VAR_TEMP
  EStopOK : BOOL ;	//auxiliary flag
  CIP : BOOL ;	//CIP Program Selected
  xTmp : BOOL ;	//Temporary Bool(free for general use)
  UnitNo : INT ;	//unit number
  UnitFB : INT ;	//unit expansion FB number
  rTmp : REAL ;	//Temporary REAL (free for general use)
  iTmp : INT ;	//Temporary INT (free for general use)
  dTmp : DINT ;	//Temporary DINT (free for general use)
END_VAR
BEGIN
NETWORK
TITLE =general

      CLR   ;
      =     #xTmp;
      =     #EStopOK;

      L     DB1950.DBW    0;
      T     #UnitNo;
      L     DB1950.DBW    2;
      T     #UnitFB;

NETWORK
TITLE =Universal value

      NOP   0;
// unv001 UnV 001 Process Status
      CALL FC    27 (
           UnitNo                   := #UnitNo,
           UnVRec                   := DB2955.unv001,
           ValExt                   := DB2955.DBD  234);

// unv002 UnV 002 Universal Value 02
      CALL FC    27 (
           UnitNo                   := #UnitNo,
           UnVRec                   := DB2955.unv002,
           ValExt                   := DB2955.DBD  362);

// RK2_KreisNr UnV 003 Circuit Number
      CALL FC    27 (
           UnitNo                   := #UnitNo,
           UnVRec                   := DB2955.RK2_KreisNr,
           ValExt                   := DB2955.DBD  490);

// RK2_Medium UnV 004 0=NIX 1=Wasser 2=Heißwasser 3=Lauge 4=Säure 5=Desi
      CALL FC    27 (
           UnitNo                   := #UnitNo,
           UnVRec                   := DB2955.RK2_Medium,
           ValExt                   := DB2955.DBD  618);

NETWORK
TITLE =special inputs

      NOP   0;
// GOA_RR2 SpI 001 GOA_RR2 Schwenkbogen Befüllblock nach RR2
      CALL FC    14 (
           UnitNo                   := #UnitNo,
           SpIRec                   := DB2951.GOA_RR2,
           SpIBit                   := I    312.0);

// RM_NI_RR2K1 SpI 002 Handklappe im Rücklauf CIP 2 hinter Befüllblock
      CALL FC    14 (
           UnitNo                   := #UnitNo,
           SpIRec                   := DB2951.RM_NI_RR2K1,
           SpIBit                   := I    312.2);

// GOA_RV2K1 SpI 003 RV2K1
      CALL FC    14 (
           UnitNo                   := #UnitNo,
           SpIRec                   := DB2951.GOA_RV2K1,
           SpIBit                   := I    276.0);

// GOA_RV2K2 SpI 004 RV2K2 zur KEG Anlage
      CALL FC    14 (
           UnitNo                   := #UnitNo,
           SpIRec                   := DB2951.GOA_RV2K2,
           SpIBit                   := I    276.1);

NETWORK
TITLE =messages

      NOP   0;
// msg001 Msg 001 Message 01
      CALL FC    16 (
           UnitNo                   := #UnitNo,
           MsgRec                   := DB2957.msg001,
           MsgBit                   := DB2957.DBX   82.7);

// msg002 Msg 002 Message 02
      CALL FC    16 (
           UnitNo                   := #UnitNo,
           MsgRec                   := DB2957.msg002,
           MsgBit                   := DB2957.DBX  142.7);

NETWORK
TITLE =unit supply

      UC    FB [#UnitFB];

NETWORK
TITLE =FW_RK1
// Act 003
// Box           : Ventilinsel 4
// Input address : I335.7
// Output address: Q335.7
      CALL FC    70 (
           UnitNo                   := #UnitNo,
           ActRec                   := DB2950.FW_RK1,
           Typ                      := 23,
           FBa                      := I    335.7,
           FBa2                     := #xTmp,
           Out                      := Q    335.7);

NETWORK
TITLE =RV2_RW
// Act 004
// Box           : VSRVK1..3
// Input address : I82.1
// Output address: Q82.1
      CALL FC    70 (
           UnitNo                   := #UnitNo,
           ActRec                   := DB2950.RV2_RW,
           Typ                      := 1,
           FBa                      := #xTmp,
           FBa2                     := I     82.1,
           Out                      := Q     82.1);

NETWORK
TITLE =RV2V1  KEG/A14 KZE
// Act 006
// Box           : VS2-BB
// Output address: Q311.1
      CALL FC    70 (
           UnitNo                   := #UnitNo,
           ActRec                   := DB2950.RV2V1,
           Typ                      := 0,
           FBa                      := #xTmp,
           FBa2                     := #xTmp,
           Out                      := Q    311.1);

NETWORK
TITLE =RV2_RS  Ventil zum Gully beim spülen vom Tank
// Act 007
// Box           : Ventilinsel 4
// Input address : I337.3
// Output address: Q337.3
      CALL FC    70 (
           UnitNo                   := #UnitNo,
           ActRec                   := DB2950.RV2_RS,
           Typ                      := 1,
           FBa                      := #xTmp,
           FBa2                     := I    337.3,
           Out                      := Q    337.3);

END_FUNCTION_BLOCK

FUNCTION_BLOCK FB 1951
TITLE =U095: CIP 2 Distribution
FAMILY : BOTEC_F1
NAME : UniE
VERSION : 1.2


VAR_TEMP
  CIP : BOOL ;	//CIP active
  UNIM : BOOL ;	//Unit Not In Maintenance
  GenRel : BOOL ;	//general OK (emergency and maintenance OK)
  EStopOK : BOOL ;	//emergency OK
  UnitNo : INT ;	//unit number
  xTmp : BOOL ;	//Temporary Bool
  iTmp : INT ;	//Temporary INT
  rTmp : REAL ;	//Temporary REAL
  dTmp : DINT ;	//Temporary DINT (free for general use)
  RetValInt : INT ;	//return value
END_VAR
BEGIN
NETWORK
TITLE =General

      SET   ;
// Simulation ---------------------------------------------------------------
      A     DB1951.DBX 1357.7;
      CC    FB  1959; // "U095Sim"
      A     DB1951.DBX   17.3;
      =     DB1951.DBX 1357.7; //Help bit for simulation

// get unit number ----------------------------------------------------------
      L     DB1950.DBW    0;
      T     #UnitNo;

// CIP ----------------------------------------------------------------------
      L     DB1951.DBD   54;
      L     0;
      <D    ;
      =     #CIP;

// emergency OK -------------------------------------------------------------
      A     DB1955.DBX   27.0; //Emergency Stop OK
      =     #EStopOK;

// Write Unit in Maintenance ------------------------------------------------

      AN    DB1951.DBX   69.7;
      =     #UNIM;

// emergency and maintenance OK ---------------------------------------------
      A     #EStopOK;
      A     #UNIM;
      =     #GenRel;

// communication ------------------------------------------------------------
      UC    FB  1955; // U095Com

NETWORK
TITLE =Universal Value

      NOP   0;

// ----------------------------------------------------------
// unv001 Process Status
// ----------------------------------------------------------
// process value to UnV
//      L     0.000000e+000
//      T     "U095UnVD".unv001.ValExt

// ----------------------------------------------------------
// unv002 Universal Value 02
// ----------------------------------------------------------
// process value to UnV
//      L     0.000000e+000
//      T     "U095UnVD".unv002.ValExt

// ----------------------------------------------------------
// RK2_KreisNr Circuit Number
// ----------------------------------------------------------
// process value to UnV
//      L     0.000000e+000
//      T     "U095UnVD".RK2_KreisNr.ValExt

// ----------------------------------------------------------
// RK2_Medium 0=NIX 1=Wasser 2=Heißwasser 3=Lauge 4=Säure 5=Desi
// ----------------------------------------------------------
// process value to UnV
//      L     0.000000e+000
//      T     "U095UnVD".RK2_Medium.ValExt

NETWORK
TITLE =Special Input

      NOP   0;

// ----------------------------------------------------------
// GOA_RR2 GOA_RR2 Schwenkbogen Befüllblock nach RR2
// ----------------------------------------------------------
//      SET
//      =     "U095SpID".GOA_RR2.EAl
//      =     "U095SpID".GOA_RR2.Pre

// ----------------------------------------------------------
// RM_NI_RR2K1 Handklappe im Rücklauf CIP 2 hinter Befüllblock
// ----------------------------------------------------------
      SET   ;
      =     DB2951.DBX  141.4;
      =     DB2951.DBX  141.5;

// ----------------------------------------------------------
// GOA_RV2K1 RV2K1
// ----------------------------------------------------------
      SET   ;
      =     DB2951.DBX  201.4;
      =     DB2951.DBX  201.5;

// ----------------------------------------------------------
// GOA_RV2K2 RV2K2 zur KEG Anlage
// ----------------------------------------------------------
      SET   ;
      =     DB2951.DBX  261.4;
      =     DB2951.DBX  261.5;

NETWORK
TITLE =Messages

      NOP   0;

// ----------------------------------------------------------
// msg001 Message 01
// ----------------------------------------------------------
      SET   ;
      R     DB2957.DBX   80.7;
      =     DB2957.DBX   81.4;

      CLR   ;
      =     DB2957.DBX   82.7;

// ----------------------------------------------------------
// msg002 Message 02
// ----------------------------------------------------------
      SET   ;
      R     DB2957.DBX  140.7;
      =     DB2957.DBX  141.4;

      CLR   ;
      =     DB2957.DBX  142.7;

NETWORK
TITLE =Sequence organisation

      CLR   ;
      =     M    122.2;

// SFM supply ----------------------------------------------------------------

// CIP Counter
//      CALL  "V2S"
//       UnitNo      :=#UnitNo
//       Value       :="U095ComD".Own.Real07
//       Enable      :=TRUE
//       Down        :=FALSE
//       OriginDetect:=0.000000e+000
//       MaxDiffPS   :=1.000000e+000
//       SFMRec      :="U095SeqD".Seq.SFM[15]
//       ValueOld    :="U095SeqD".Seq.User.Real15

// sequencer ----------------------------------------------------------------
      A     DB1953.DBX   43.1;
      S     DB1953.DBX   97.3;

      CALL FC    40 (
           UnitNo                   := #UnitNo);

NETWORK
TITLE =Auto / Manual

      SET   ;
      AN    M    122.2;
      JC    MODE;
      AN    M    120.1;
      =     DB2950.DBX  265.4;
      =     DB2950.DBX  345.4;
      =     DB2950.DBX  505.4;
      =     DB2950.DBX  585.4;


MODE: SET   ;


NETWORK
TITLE =FW_RK1
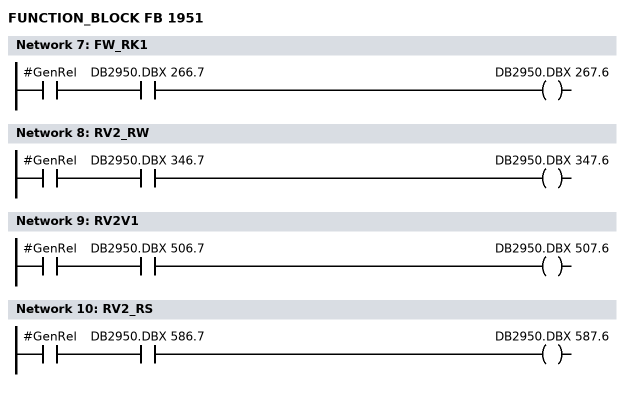

      A     #GenRel;
      A     DB2950.DBX  266.7;
      =     DB2950.DBX  267.6;
NETWORK
TITLE =RV2_RW

      A     #GenRel;
      A     DB2950.DBX  346.7;
      =     DB2950.DBX  347.6;

NETWORK
TITLE =RV2V1

      A     #GenRel;
      A     DB2950.DBX  506.7;
      =     DB2950.DBX  507.6;
NETWORK
TITLE =RV2_RS


      A     #GenRel;
      A     DB2950.DBX  586.7;
      =     DB2950.DBX  587.6;
END_FUNCTION_BLOCK

FUNCTION_BLOCK FB 1960
TITLE =U096: CIP 3 Distribution
FAMILY : BOTEC_F1
NAME : UniA
VERSION : 2.1


VAR_TEMP
  EStopOK : BOOL ;	//auxiliary flag
  CIP : BOOL ;	//CIP Program Selected
  xTmp : BOOL ;	//Temporary Bool(free for general use)
  UnitNo : INT ;	//unit number
  UnitFB : INT ;	//unit expansion FB number
  rTmp : REAL ;	//Temporary REAL (free for general use)
  iTmp : INT ;	//Temporary INT (free for general use)
  dTmp : DINT ;	//Temporary DINT (free for general use)
END_VAR
BEGIN
NETWORK
TITLE =general

      CLR   ;
      =     #xTmp;
      =     #EStopOK;

      L     DB1960.DBW    0;
      T     #UnitNo;
      L     DB1960.DBW    2;
      T     #UnitFB;

NETWORK
TITLE =Universal value

      NOP   0;
// unv001 UnV 001 Process Status
      CALL FC    27 (
           UnitNo                   := #UnitNo,
           UnVRec                   := DB2965.unv001,
           ValExt                   := DB2965.DBD  234);

// unv002 UnV 002 Universal Value 02
      CALL FC    27 (
           UnitNo                   := #UnitNo,
           UnVRec                   := DB2965.unv002,
           ValExt                   := DB2965.DBD  362);

// RK3_KreisNr UnV 003 Circuit Number
      CALL FC    27 (
           UnitNo                   := #UnitNo,
           UnVRec                   := DB2965.RK3_KreisNr,
           ValExt                   := DB2965.DBD  490);

// RK3_Medium UnV 004 0=NIX 1=Wasser 2=Heißwasser 3=Lauge 4=Säure 5=Desi
      CALL FC    27 (
           UnitNo                   := #UnitNo,
           UnVRec                   := DB2965.RK3_Medium,
           ValExt                   := DB2965.DBD  618);

NETWORK
TITLE =special inputs

      NOP   0;
// RK3_I_Bereit SpI 001 Das Reinigungs Programm ist gestartet und läuft "1"= Läuft  "0"=AUS
      CALL FC    14 (
           UnitNo                   := #UnitNo,
           SpIRec                   := DB2961.RK3_I_Bereit,
           SpIBit                   := DB304.DBX   30.0);

// RK3_I_VL_Ein SpI 002 Medium wird angefordert (Reinigungs Vorlauf EIN) "1"=VorlaufPumpe an "0"AUS
      CALL FC    14 (
           UnitNo                   := #UnitNo,
           SpIRec                   := DB2961.RK3_I_VL_Ein,
           SpIBit                   := DB304.DBX   30.1);

// RK3_I_RL_Ein SpI 003 Medium wird zurückgepumpt "1" RücklaufPumpe an "0"=AUS
      CALL FC    14 (
           UnitNo                   := #UnitNo,
           SpIRec                   := DB2961.RK3_I_RL_Ein,
           SpIBit                   := DB304.DBX   30.2);

// RK3_I_Leer SpI 004 Der zu Reinigende Anlagenteil ist leer."1"=leer "0"=nicht leer
      CALL FC    14 (
           UnitNo                   := #UnitNo,
           SpIRec                   := DB2961.RK3_I_Leer,
           SpIBit                   := DB304.DBX   30.3);

// RK3_I_Stop SpI 005 Stop interner Fehler Pumpen anhalten Reinigungszeit anhalten "1" STOP  "0"= OK
      CALL FC    14 (
           UnitNo                   := #UnitNo,
           SpIRec                   := DB2961.RK3_I_Stop,
           SpIBit                   := DB304.DBX   30.4);

// RK3_I_SK_RM SpI 006 Bypassventil ist angesteuert und offen
      CALL FC    14 (
           UnitNo                   := #UnitNo,
           SpIRec                   := DB2961.RK3_I_SK_RM,
           SpIBit                   := DB304.DBX   30.7);

NETWORK
TITLE =messages

      NOP   0;
// msg001 Msg 001 Message 01
      CALL FC    16 (
           UnitNo                   := #UnitNo,
           MsgRec                   := DB2967.msg001,
           MsgBit                   := DB2967.DBX   82.7);

// msg002 Msg 002 Message 02
      CALL FC    16 (
           UnitNo                   := #UnitNo,
           MsgRec                   := DB2967.msg002,
           MsgBit                   := DB2967.DBX  142.7);

NETWORK
TITLE =unit supply

      UC    FB [#UnitFB];

NETWORK
TITLE =RV3_ST
// Act 004
// Box           : VSRVK1..3
// Input address : I82.2
// Output address: Q82.2
      CALL FC    70 (
           UnitNo                   := #UnitNo,
           ActRec                   := DB2960.RV3_ST,
           Typ                      := 1,
           FBa                      := #xTmp,
           FBa2                     := I     82.2,
           Out                      := Q     82.2);

NETWORK
TITLE =K3_VNI_RSTP  STOP TU AN VNI MELDEN
// Act 004
// Box           : S8 U8.2
// Output address: Q42.0
      CALL FC    70 (
           UnitNo                   := #UnitNo,
           ActRec                   := DB2960.K3_VNI_RSTP,
           Typ                      := 0,
           FBa                      := #xTmp,
           FBa2                     := #xTmp,
           Out                      := Q     42.0);

NETWORK
TITLE =K3_VNI_RMW  MEDIENWECHSEL AN VNI MELDEN
// Act 005
// Box           : S8 U8.2
// Output address: Q42.1
      CALL FC    70 (
           UnitNo                   := #UnitNo,
           ActRec                   := DB2960.K3_VNI_RMW,
           Typ                      := 0,
           FBa                      := #xTmp,
           FBa2                     := #xTmp,
           Out                      := Q     42.1);

NETWORK
TITLE =K3_VNI_REND  ENDE MELDUNG AN VNI
// Act 006
// Box           : S8 U8.2
// Output address: Q42.2
      CALL FC    70 (
           UnitNo                   := #UnitNo,
           ActRec                   := DB2960.K3_VNI_REND,
           Typ                      := 0,
           FBa                      := #xTmp,
           FBa2                     := #xTmp,
           Out                      := Q     42.2);

NETWORK
TITLE =K3_VNI_RHL  MELDUNG HEISSLAUGE AN VNI
// Act 007
// Box           : S8 U8.2
// Output address: Q42.3
      CALL FC    70 (
           UnitNo                   := #UnitNo,
           ActRec                   := DB2960.K3_VNI_RHL,
           Typ                      := 0,
           FBa                      := #xTmp,
           FBa2                     := #xTmp,
           Out                      := Q     42.3);

NETWORK
TITLE =K3_VNI_RBTR  BETRIEBSMELDUNG CIP AN VNI
// Act 008
// Box           : S8 U8.2
// Output address: Q42.4
      CALL FC    70 (
           UnitNo                   := #UnitNo,
           ActRec                   := DB2960.K3_VNI_RBTR,
           Typ                      := 0,
           FBa                      := #xTmp,
           FBa2                     := #xTmp,
           Out                      := Q     42.4);

NETWORK
TITLE =K3_VNI_WASSER_OK  WASSER OK AN VNI
// Act 009
// Box           : S8 U8.2
// Output address: Q42.5
      CALL FC    70 (
           UnitNo                   := #UnitNo,
           ActRec                   := DB2960.K3_VNI_WASSER_OK,
           Typ                      := 0,
           FBa                      := #xTmp,
           FBa2                     := #xTmp,
           Out                      := Q     42.5);

NETWORK
TITLE =RK3_Bereit  Die CIP Station hat gestatet "0"=AUS "1"=gestartet
// Act 010
// Box           : Sirup
// Output address: DB_SEND_DOEHLER.RK3.Bereit
      CALL FC    70 (
           UnitNo                   := #UnitNo,
           ActRec                   := DB2960.RK3_Bereit,
           Typ                      := 0,
           FBa                      := #xTmp,
           FBa2                     := #xTmp,
           Out                      := DB404.DBX   30.0);

NETWORK
TITLE =RK3_Stop  Stop Pumpen anhalten "0"Ok" 1"=Stop
// Act 011
// Box           : Sirup
// Output address: DB_SEND_DOEHLER.RK3.Stop
      CALL FC    70 (
           UnitNo                   := #UnitNo,
           ActRec                   := DB2960.RK3_Stop,
           Typ                      := 0,
           FBa                      := #xTmp,
           FBa2                     := #xTmp,
           Out                      := DB404.DBX   30.1);

NETWORK
TITLE =RK3_MED  Medienwechsel der CIP
// Act 012
// Box           : Sirup
// Output address: DB_SEND_DOEHLER.RK3.MED
      CALL FC    70 (
           UnitNo                   := #UnitNo,
           ActRec                   := DB2960.RK3_MED,
           Typ                      := 0,
           FBa                      := #xTmp,
           FBa2                     := #xTmp,
           Out                      := DB404.DBX   30.2);

NETWORK
TITLE =RK3_ENDE  Ende der Reinigung
// Act 013
// Box           : Sirup
// Output address: DB_SEND_DOEHLER.RK3.ENDE
      CALL FC    70 (
           UnitNo                   := #UnitNo,
           ActRec                   := DB2960.RK3_ENDE,
           Typ                      := 0,
           FBa                      := #xTmp,
           FBa2                     := #xTmp,
           Out                      := DB404.DBX   30.3);

NETWORK
TITLE =RK3_Bypass  CIP Bypass
// Act 014
// Box           : Sirup
// Output address: DB_SEND_DOEHLER.RK3.Bypass
      CALL FC    70 (
           UnitNo                   := #UnitNo,
           ActRec                   := DB2960.RK3_Bypass,
           Typ                      := 0,
           FBa                      := #xTmp,
           FBa2                     := #xTmp,
           Out                      := DB404.DBX   30.4);

NETWORK
TITLE =SR1_RR3  SR1 RR3 CIP Rücklaufventil RR3SR1
// Act 015
// Box           : VS-RRA
// Input address : I200.7
// Output address: Q200.7
      CALL FC    70 (
           UnitNo                   := #UnitNo,
           ActRec                   := DB2960.SR1_RR3,
           Typ                      := 1,
           FBa                      := #xTmp,
           FBa2                     := I    200.7,
           Out                      := Q    200.7);

NETWORK
TITLE =SR2_RR3  SR2 RR3 CIP Rücklaufventil RR3SR2
// Act 016
// Box           : VS-RRA
// Input address : I201.1
// Output address: Q201.1
      CALL FC    70 (
           UnitNo                   := #UnitNo,
           ActRec                   := DB2960.SR2_RR3,
           Typ                      := 1,
           FBa                      := #xTmp,
           FBa2                     := I    201.1,
           Out                      := Q    201.1);

NETWORK
TITLE =RV3_RS  Ventil zum Gully beim spülen vom Tank
// Act 019
// Box           : Ventilinsel 4
// Input address : I337.4
// Output address: Q337.4
      CALL FC    70 (
           UnitNo                   := #UnitNo,
           ActRec                   := DB2960.RV3_RS,
           Typ                      := 1,
           FBa                      := #xTmp,
           FBa2                     := I    337.4,
           Out                      := Q    337.4);

END_FUNCTION_BLOCK

FUNCTION_BLOCK FB 1961
TITLE =U096: CIP 3 Distribution
FAMILY : BOTEC_F1
NAME : UniE
VERSION : 1.2


VAR_TEMP
  CIP : BOOL ;	//CIP active
  UNIM : BOOL ;	//Unit Not In Maintenance
  GenRel : BOOL ;	//general OK (emergency and maintenance OK)
  EStopOK : BOOL ;	//emergency OK
  UnitNo : INT ;	//unit number
  xTmp : BOOL ;	//Temporary Bool
  iTmp : INT ;	//Temporary INT
  rTmp : REAL ;	//Temporary REAL
  dTmp : DINT ;	//Temporary DINT (free for general use)
  RetValInt : INT ;	//return value
END_VAR
BEGIN
NETWORK
TITLE =General

      SET   ;
// Simulation ---------------------------------------------------------------
      A     DB1961.DBX 1357.7;
      CC    FB  1969; // "U096Sim"
      A     DB1961.DBX   17.3;
      =     DB1961.DBX 1357.7; //Help bit for simulation

// get unit number ----------------------------------------------------------
      L     DB1960.DBW    0;
      T     #UnitNo;

// CIP ----------------------------------------------------------------------
      L     DB1961.DBD   54;
      L     0;
      <D    ;
      =     #CIP;

// emergency OK -------------------------------------------------------------
      A     DB1965.DBX   27.0; //Emergency Stop OK
      =     #EStopOK;

// Write Unit in Maintenance ------------------------------------------------

      AN    DB1961.DBX   69.7;
      =     #UNIM;

// emergency and maintenance OK ---------------------------------------------
      A     #EStopOK;
      A     #UNIM;
      =     #GenRel;

// communication ------------------------------------------------------------
      UC    FB  1965; // U096Com

NETWORK
TITLE =Universal Value

      NOP   0;

// ----------------------------------------------------------
// unv001 Process Status
// ----------------------------------------------------------
// process value to UnV
//      L     0.000000e+000
//      T     "U096UnVD".unv001.ValExt

// ----------------------------------------------------------
// unv002 Universal Value 02
// ----------------------------------------------------------
// process value to UnV
//      L     0.000000e+000
//      T     "U096UnVD".unv002.ValExt

// ----------------------------------------------------------
// RK3_KreisNr Circuit Number
// ----------------------------------------------------------
// process value to UnV
//      L     0.000000e+000
//      T     "U096UnVD".RK3_KreisNr.ValExt

// ----------------------------------------------------------
// RK3_Medium 0=NIX 1=Wasser 2=Heißwasser 3=Lauge 4=Säure 5=Desi
// ----------------------------------------------------------
// process value to UnV
//      L     0.000000e+000
//      T     "U096UnVD".RK3_Medium.ValExt

NETWORK
TITLE =Special Input

      NOP   0;

// ----------------------------------------------------------
// RK3_I_Bereit Das Reinigungs Programm ist gestartet und läuft "1"= Läuft  "0"=AUS
// ----------------------------------------------------------
      CLR   ;
      =     DB2961.DBX   81.4;
      =     DB2961.DBX   81.5;

// ----------------------------------------------------------
// RK3_I_VL_Ein Medium wird angefordert (Reinigungs Vorlauf EIN) "1"=VorlaufPumpe an "0"AUS
// ----------------------------------------------------------
      CLR   ;
      =     DB2961.DBX  141.4;
      =     DB2961.DBX  141.5;

// ----------------------------------------------------------
// RK3_I_RL_Ein Medium wird zurückgepumpt "1" RücklaufPumpe an "0"=AUS
// ----------------------------------------------------------
      CLR   ;
      =     DB2961.DBX  201.4;
      =     DB2961.DBX  201.5;

// ----------------------------------------------------------
// RK3_I_Leer Der zu Reinigende Anlagenteil ist leer."1"=leer "0"=nicht leer
// ----------------------------------------------------------
      CLR   ;
      =     DB2961.DBX  261.4;
      =     DB2961.DBX  261.5;

// ----------------------------------------------------------
// RK3_I_Stop Stop interner Fehler Pumpen anhalten Reinigungszeit anhalten "1" STOP  "0"= OK
// ----------------------------------------------------------
      CLR   ;
      =     DB2961.DBX  321.4;
      =     DB2961.DBX  321.5;

// ----------------------------------------------------------
// RK3_I_SK_RM Bypassventil ist angesteuert und offen
// ----------------------------------------------------------
      CLR   ;
      =     DB2961.DBX  381.4;
      =     DB2961.DBX  381.5;

NETWORK
TITLE =Messages

      NOP   0;

// ----------------------------------------------------------
// msg001 Message 01
// ----------------------------------------------------------
      SET   ;
      R     DB2967.DBX   80.7;
      =     DB2967.DBX   81.4;

      CLR   ;
      =     DB2967.DBX   82.7;

// ----------------------------------------------------------
// msg002 Message 02
// ----------------------------------------------------------
      SET   ;
      R     DB2967.DBX  140.7;
      =     DB2967.DBX  141.4;

      CLR   ;
      =     DB2967.DBX  142.7;

NETWORK
TITLE =Sequence organisation

      CLR   ;
      =     M    122.2;

// SFM supply ----------------------------------------------------------------

      CALL FC    29 (
           UnitNo                   := #UnitNo,
           Value                    := DB1965.DBD   54,
           Enable                   := TRUE,
           Down                     := FALSE,
           OriginDetect             := 0.000000e+000,
           MaxDiffPS                := 1.000000e+000,
           SFMRec                   := DB1961.Seq.SFM[15],
           ValueOld                 := DB1961.DBD 1418);

// sequencer ----------------------------------------------------------------
      A     DB1963.DBX   43.1;
      S     DB1963.DBX   97.3;

      CALL FC    40 (
           UnitNo                   := #UnitNo);

NETWORK
TITLE =Auto / Manual

      SET   ;
      AN    M    122.2;
      JC    MODE;
      AN    M    120.1;

// assign actuator mode
      AN    M    120.1;
      =     DB2960.DBX  185.4;
      =     DB2960.DBX  265.4;
      =     DB2960.DBX  345.4;
      =     DB2960.DBX  425.4;
      =     DB2960.DBX  505.4;
      =     DB2960.DBX  585.4;
      =     DB2960.DBX  665.4;
      =     DB2960.DBX  745.4;
      =     DB2960.DBX  825.4;
      =     DB2960.DBX  905.4;
      =     DB2960.DBX  985.4;
      =     DB2960.DBX 1065.4;
      =     DB2960.DBX 1145.4;
      =     DB2960.DBX 1225.4;
      =     DB2960.DBX 1305.4;
      =     DB2960.DBX 1545.4;

MODE: SET   ;

NETWORK
TITLE =RV3_ST
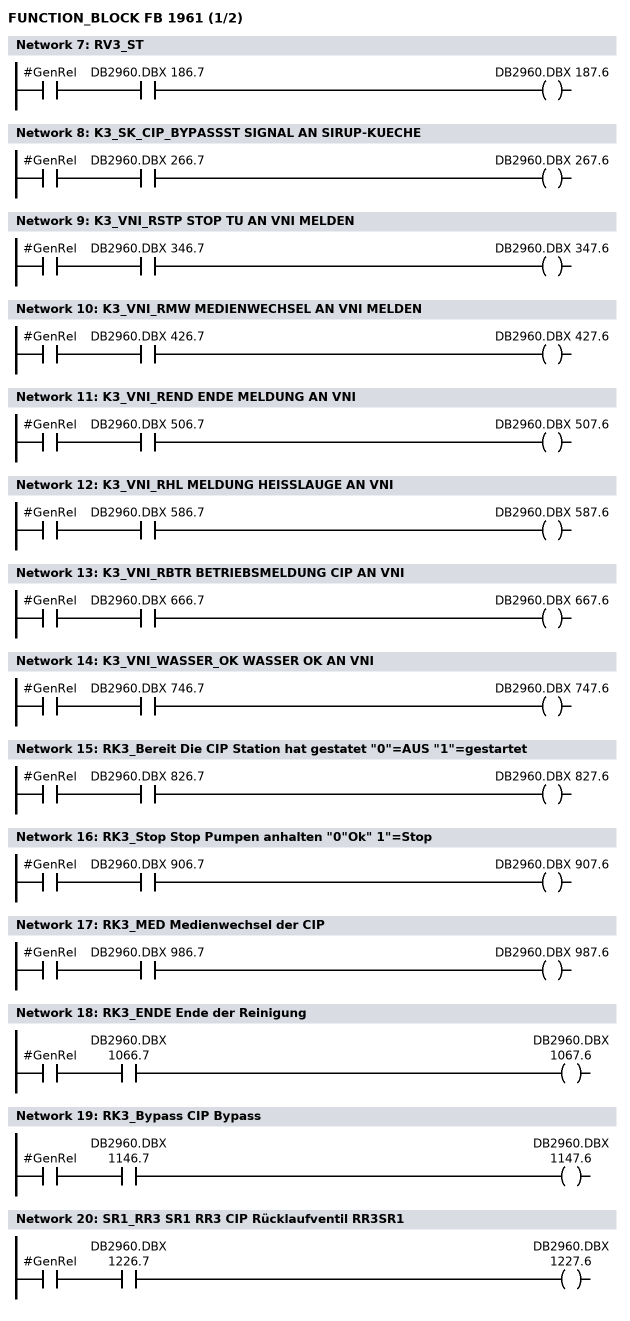

      A     #GenRel;
      A     DB2960.DBX  186.7;
      =     DB2960.DBX  187.6;
NETWORK
TITLE =K3_SK_CIP_BYPASSST SIGNAL AN SIRUP-KUECHE

      A     #GenRel;
      A     DB2960.DBX  266.7;
      =     DB2960.DBX  267.6;
NETWORK
TITLE =K3_VNI_RSTP STOP TU AN VNI MELDEN

      A     #GenRel;
      A     DB2960.DBX  346.7;
      =     DB2960.DBX  347.6;
NETWORK
TITLE =K3_VNI_RMW MEDIENWECHSEL AN VNI MELDEN

      A     #GenRel;
      A     DB2960.DBX  426.7;
      =     DB2960.DBX  427.6;
NETWORK
TITLE =K3_VNI_REND ENDE MELDUNG AN VNI

      A     #GenRel;
      A     DB2960.DBX  506.7;
      =     DB2960.DBX  507.6;
NETWORK
TITLE =K3_VNI_RHL MELDUNG HEISSLAUGE AN VNI

      A     #GenRel;
      A     DB2960.DBX  586.7;
      =     DB2960.DBX  587.6;
NETWORK
TITLE =K3_VNI_RBTR BETRIEBSMELDUNG CIP AN VNI

      A     #GenRel;
      A     DB2960.DBX  666.7;
      =     DB2960.DBX  667.6;
NETWORK
TITLE =K3_VNI_WASSER_OK WASSER OK AN VNI

      A     #GenRel;
      A     DB2960.DBX  746.7;
      =     DB2960.DBX  747.6;
NETWORK
TITLE =RK3_Bereit Die CIP Station hat gestatet "0"=AUS "1"=gestartet

      A     #GenRel;
      A     DB2960.DBX  826.7;
      =     DB2960.DBX  827.6;
NETWORK
TITLE =RK3_Stop Stop Pumpen anhalten "0"Ok" 1"=Stop

      A     #GenRel;
      A     DB2960.DBX  906.7;
      =     DB2960.DBX  907.6;
NETWORK
TITLE =RK3_MED Medienwechsel der CIP

      A     #GenRel;
      A     DB2960.DBX  986.7;
      =     DB2960.DBX  987.6;
NETWORK
TITLE =RK3_ENDE Ende der Reinigung

      A     #GenRel;
      A     DB2960.DBX 1066.7;
      =     DB2960.DBX 1067.6;
NETWORK
TITLE =RK3_Bypass CIP Bypass

      A     #GenRel;
      A     DB2960.DBX 1146.7;
      =     DB2960.DBX 1147.6;
NETWORK
TITLE =SR1_RR3 SR1 RR3 CIP Rücklaufventil RR3SR1

      A     #GenRel;
      A     DB2960.DBX 1226.7;
      =     DB2960.DBX 1227.6;
NETWORK
TITLE =SR2_RR3 SR2 RR3 CIP Rücklaufventil RR3SR2
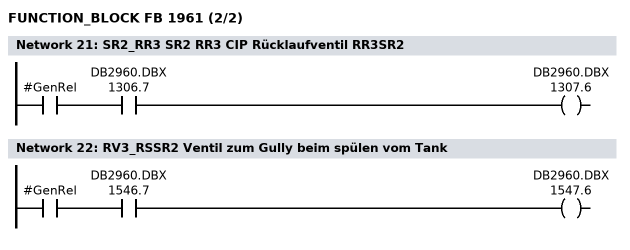

      A     #GenRel;
      A     DB2960.DBX 1306.7;
      =     DB2960.DBX 1307.6;
NETWORK
TITLE =RV3_RSSR2 Ventil zum Gully beim spülen vom Tank

      A     #GenRel;
      A     DB2960.DBX 1546.7;
      =     DB2960.DBX 1547.6;
END_FUNCTION_BLOCK

FUNCTION_BLOCK FB 1980
TITLE =U098: General Syrup Room
FAMILY : BOTEC_F1
NAME : UniA
VERSION : 2.1


VAR_TEMP
  EStopOK : BOOL ;	//auxiliary flag
  CIP : BOOL ;	//CIP Program Selected
  xTmp : BOOL ;	//Temporary Bool(free for general use)
  UnitNo : INT ;	//unit number
  UnitFB : INT ;	//unit expansion FB number
  rTmp : REAL ;	//Temporary REAL (free for general use)
  iTmp : INT ;	//Temporary INT (free for general use)
  dTmp : DINT ;	//Temporary DINT (free for general use)
END_VAR
BEGIN
NETWORK
TITLE =general

      CLR   ;
      =     #xTmp;
      =     #EStopOK;

      L     DB1980.DBW    0;
      T     #UnitNo;
      L     DB1980.DBW    2;
      T     #UnitFB;

NETWORK
TITLE =analog inputs

      NOP   0;
// IW518 AnI 001 Produkttemp. Erhitzer
      CALL FC    24 (
           UnitNo                   := #UnitNo,
           AnIRec                   := DB2983._PIW518,
           ValPer                   := IW   518);

// IW520 AnI 002 Erhitzungsregelung Heisswasser
      CALL FC    24 (
           UnitNo                   := #UnitNo,
           AnIRec                   := DB2983._PIW520,
           ValPer                   := IW   520);

// IW522 AnI 003 Produkttemp. Kühler
      CALL FC    24 (
           UnitNo                   := #UnitNo,
           AnIRec                   := DB2983._PIW522,
           ValPer                   := IW   522);

// IW524 AnI 004 Produkteintrittstemp.
      CALL FC    24 (
           UnitNo                   := #UnitNo,
           AnIRec                   := DB2983._PIW524,
           ValPer                   := IW   524);

NETWORK
TITLE =Universal value

      NOP   0;
// unv001 UnV 001 Process Status
      CALL FC    27 (
           UnitNo                   := #UnitNo,
           UnVRec                   := DB2985.unv001,
           ValExt                   := DB2985.DBD  234);

// unv002 UnV 002 Universal Value 02
      CALL FC    27 (
           UnitNo                   := #UnitNo,
           UnVRec                   := DB2985.unv002,
           ValExt                   := DB2985.DBD  362);

// IW532 UnV 003 Contents Zitronensäuretank
      CALL FC    27 (
           UnitNo                   := #UnitNo,
           UnVRec                   := DB2985._PIW532,
           ValExt                   := DB2985.DBD  490);

// WAS_Wasser_Druck UnV 004 Water Pressure in Bar
      CALL FC    27 (
           UnitNo                   := #UnitNo,
           UnVRec                   := DB2985.WAS_Wasser_Druck,
           ValExt                   := DB2985.DBD  618);

NETWORK
TITLE =special inputs

      NOP   0;
// NI_RR_SIRUPWASSER SpI 001 PANEEL SIRUPKUECHE (???)
      CALL FC    14 (
           UnitNo                   := #UnitNo,
           SpIRec                   := DB2981.NI_RR_SIRUPWASSER,
           SpIBit                   := I    102.7);

// KZE_FREIGABE_CIP SpI 002 SIGNAL VON SCHMIDT KZE SK
      CALL FC    14 (
           UnitNo                   := #UnitNo,
           SpIRec                   := DB2981.KZE_FREIGABE_CIP,
           SpIBit                   := I     65.1);

// KZE_KEIN_STOP SpI 003 SIGNAL VON SCHMIDT KZE SK
      CALL FC    14 (
           UnitNo                   := #UnitNo,
           SpIRec                   := DB2981.KZE_KEIN_STOP,
           SpIBit                   := I     65.2);

// KZE_INTERNE_REINIGUNG SpI 004 SIGNAL VON SCHMIDT KZE SK
      CALL FC    14 (
           UnitNo                   := #UnitNo,
           SpIRec                   := DB2981.KZE_INTERNE_REINIGUNG,
           SpIBit                   := I     65.3);

// KZE_TANK_LEERMELDUNG SpI 005 SIGNAL VON SCHMIDT KZE SK
      CALL FC    14 (
           UnitNo                   := #UnitNo,
           SpIRec                   := DB2981.KZE_TANK_LEERMELDUNG,
           SpIBit                   := I     65.4);

// KZE_FREIGABE_VORLAUF SpI 006 SIGNAL VON SCHMIDT KZE SK
      CALL FC    14 (
           UnitNo                   := #UnitNo,
           SpIRec                   := DB2981.KZE_FREIGABE_VORLAUF,
           SpIBit                   := I     65.5);

// LDT_START_MOLCH_S1 SpI 007 STARTTASTER AB SIRUPKUECHE
      CALL FC    14 (
           UnitNo                   := #UnitNo,
           SpIRec                   := DB2981.LDT_START_MOLCH_S1,
           SpIBit                   := I     66.2);

// LANG_STOER_DOSIERUNG SpI 008 RUECKMELDUNG VON LANG AN TU
      CALL FC    14 (
           UnitNo                   := #UnitNo,
           SpIRec                   := DB2981.LANG_STOER_DOSIERUNG,
           SpIBit                   := I     40.3);

// LiveBit SpI 009
      CALL FC    14 (
           UnitNo                   := #UnitNo,
           SpIRec                   := DB2981.LiveBit,
           SpIBit                   := DB304.DBX    0.0);

NETWORK
TITLE =messages

      NOP   0;
// msg001 Msg 001 Message 01
      CALL FC    16 (
           UnitNo                   := #UnitNo,
           MsgRec                   := DB2987.msg001,
           MsgBit                   := DB2987.DBX   82.7);

// msg002 Msg 002 Message 02
      CALL FC    16 (
           UnitNo                   := #UnitNo,
           MsgRec                   := DB2987.msg002,
           MsgBit                   := DB2987.DBX  142.7);

NETWORK
TITLE =unit supply

      UC    FB [#UnitFB];

NETWORK
TITLE =KZE_RBTR  SIGNAL AN SCHMIDT KZE SK
// Act 001
// Box           : S8 U8.2
// Output address: Q122.0
      CALL FC    70 (
           UnitNo                   := #UnitNo,
           ActRec                   := DB2980.KZE_RBTR,
           Typ                      := 0,
           FBa                      := #xTmp,
           FBa2                     := #xTmp,
           Out                      := Q    122.0);

NETWORK
TITLE =KZE_RMW  SIGNAL AN SCHMIDT KZE SK
// Act 002
// Box           : S8 U8.2
// Output address: Q122.1
      CALL FC    70 (
           UnitNo                   := #UnitNo,
           ActRec                   := DB2980.KZE_RMW,
           Typ                      := 0,
           FBa                      := #xTmp,
           FBa2                     := #xTmp,
           Out                      := Q    122.1);

NETWORK
TITLE =KZE_RSTP  SIGNAL AN SCHMIDT KZE SK
// Act 003
// Box           : S8 U8.2
// Output address: Q122.2
      CALL FC    70 (
           UnitNo                   := #UnitNo,
           ActRec                   := DB2980.KZE_RSTP,
           Typ                      := 0,
           FBa                      := #xTmp,
           FBa2                     := #xTmp,
           Out                      := Q    122.2);

NETWORK
TITLE =KZE_REND  SIGNAL AN SCHMIDT KZE SK
// Act 004
// Box           : S8 U8.2
// Output address: Q122.3
      CALL FC    70 (
           UnitNo                   := #UnitNo,
           ActRec                   := DB2980.KZE_REND,
           Typ                      := 0,
           FBa                      := #xTmp,
           FBa2                     := #xTmp,
           Out                      := Q    122.3);

NETWORK
TITLE =KZE_MANNLOCH_OEFFNEN  SIGNAL AN SCHMIDT KZE SK
// Act 005
// Box           : S8 U8.2
// Output address: Q122.4
      CALL FC    70 (
           UnitNo                   := #UnitNo,
           ActRec                   := DB2980.KZE_MANNLOCH_OEFFNEN,
           Typ                      := 0,
           FBa                      := #xTmp,
           FBa2                     := #xTmp,
           Out                      := Q    122.4);

NETWORK
TITLE =LA_S1_MOLCH_START  LAMPE LDT AB SIRUPKUECHE
// Act 006
// Box           : S8 U8.2
// Output address: Q122.7
      CALL FC    70 (
           UnitNo                   := #UnitNo,
           ActRec                   := DB2980.LA_S1_MOLCH_START,
           Typ                      := 0,
           FBa                      := #xTmp,
           FBa2                     := #xTmp,
           Out                      := Q    122.7);

NETWORK
TITLE =Act007 spare
// Act 007
// Box           : S8 U8.2
// Output address: Q123.0
      CALL FC    70 (
           UnitNo                   := #UnitNo,
           ActRec                   := DB2980.Act007,
           Typ                      := 0,
           FBa                      := #xTmp,
           FBa2                     := #xTmp,
           Out                      := #xTmp);

NETWORK
TITLE =Act008 spare
// Act 008
// Box           : S8 U8.2
// Output address: Q123.7
      CALL FC    70 (
           UnitNo                   := #UnitNo,
           ActRec                   := DB2980.Act008,
           Typ                      := 0,
           FBa                      := #xTmp,
           FBa2                     := #xTmp,
           Out                      := #xTmp);

END_FUNCTION_BLOCK

FUNCTION_BLOCK FB 1981
TITLE =U098: General Syrup Room
FAMILY : BOTEC_F1
NAME : UniE
VERSION : 1.2


VAR_TEMP
  CIP : BOOL ;	//CIP active
  UNIM : BOOL ;	//Unit Not In Maintenance
  GenRel : BOOL ;	//general OK (emergency and maintenance OK)
  EStopOK : BOOL ;	//emergency OK
  UnitNo : INT ;	//unit number
  xTmp : BOOL ;	//Temporary Bool
  iTmp : INT ;	//Temporary INT
  rTmp : REAL ;	//Temporary REAL
  dTmp : DINT ;	//Temporary DINT (free for general use)
  RetValInt : INT ;	//return value
END_VAR
BEGIN
NETWORK
TITLE =General

      SET   ;
// Simulation ---------------------------------------------------------------
      A     DB1981.DBX 1357.7;
      CC    FB  1989; // "U098Sim"
      A     DB1981.DBX   17.3;
      =     DB1981.DBX 1357.7; //Help bit for simulation

// get unit number ----------------------------------------------------------
      L     DB1980.DBW    0;
      T     #UnitNo;

// CIP ----------------------------------------------------------------------
      L     DB1981.DBD   54;
      L     0;
      <D    ;
      =     #CIP;

// emergency OK -------------------------------------------------------------
      A     DB1985.DBX   27.0; //Emergency Stop OK
      =     #EStopOK;

// Write Unit in Maintenance ------------------------------------------------

      AN    DB1981.DBX   69.7;
      =     #UNIM;

// emergency and maintenance OK ---------------------------------------------
      A     #EStopOK;
      A     #UNIM;
      =     #GenRel;

// communication ------------------------------------------------------------
      UC    FB  1985; // U098Com

NETWORK
TITLE =Analog Inputs

      NOP   0;

// ----------------------------------------------------------
// PIW518 Produkttemp. Erhitzer
// ----------------------------------------------------------
      L     DB1981.DBD 1118; // !!! insert correct SFM !!!
      T     DB2983.DBD  238;

      SET   ;
      =     DB2983.DBX  141.5;

// ----------------------------------------------------------
// PIW520 Erhitzungsregelung Heisswasser
// ----------------------------------------------------------
      L     DB1981.DBD 1118; // !!! insert correct SFM !!!
      T     DB2983.DBD  358;

      SET   ;
      =     DB2983.DBX  261.5;

// ----------------------------------------------------------
// PIW522 Produkttemp. Kühler
// ----------------------------------------------------------
      L     DB1981.DBD 1118; // !!! insert correct SFM !!!
      T     DB2983.DBD  478;

      SET   ;
      =     DB2983.DBX  381.5;

// ----------------------------------------------------------
// PIW524 Produkteintrittstemp.
// ----------------------------------------------------------
      L     DB1981.DBD 1118; // !!! insert correct SFM !!!
      T     DB2983.DBD  598;

      SET   ;
      =     DB2983.DBX  501.5;

NETWORK
TITLE =Universal Value

      NOP   0;

// ----------------------------------------------------------
// unv001 Process Status
// ----------------------------------------------------------
// process value to UnV
//      L     0.000000e+000
//      T     "U098UnVD".unv001.ValExt

// ----------------------------------------------------------
// unv002 Universal Value 02
// ----------------------------------------------------------
// process value to UnV
//      L     0.000000e+000
//      T     "U098UnVD".unv002.ValExt

// ----------------------------------------------------------
// PIW532 Contents Zitronensäuretank
// ----------------------------------------------------------
// process value to UnV
//      L     0.000000e+000
//      T     "U098UnVD".PIW532.ValExt

// ----------------------------------------------------------
// WAS_Wasser_Druck Water Pressure in Bar
// ----------------------------------------------------------
// process value to UnV
//      L     0.000000e+000
//      T     "U098UnVD".WAS_Wasser_Druck.ValExt

NETWORK
TITLE =Special Input

      NOP   0;

// ----------------------------------------------------------
// NI_RR_SIRUPWASSER PANEEL SIRUPKUECHE (???)
// ----------------------------------------------------------
      SET   ;
      =     DB2981.DBX   81.4;
      =     DB2981.DBX   81.5;

// ----------------------------------------------------------
// KZE_FREIGABE_CIP SIGNAL VON SCHMIDT KZE SK
// ----------------------------------------------------------
      SET   ;
      =     DB2981.DBX  141.4;
      =     DB2981.DBX  141.5;

// ----------------------------------------------------------
// KZE_KEIN_STOP SIGNAL VON SCHMIDT KZE SK
// ----------------------------------------------------------
      SET   ;
      =     DB2981.DBX  201.4;
      =     DB2981.DBX  201.5;

// ----------------------------------------------------------
// KZE_INTERNE_REINIGUNG SIGNAL VON SCHMIDT KZE SK
// ----------------------------------------------------------
      SET   ;
      =     DB2981.DBX  261.4;
      =     DB2981.DBX  261.5;

// ----------------------------------------------------------
// KZE_TANK_LEERMELDUNG SIGNAL VON SCHMIDT KZE SK
// ----------------------------------------------------------
      SET   ;
      =     DB2981.DBX  321.4;
      =     DB2981.DBX  321.5;

// ----------------------------------------------------------
// KZE_FREIGABE_VORLAUF SIGNAL VON SCHMIDT KZE SK
// ----------------------------------------------------------
      SET   ;
      =     DB2981.DBX  381.4;
      =     DB2981.DBX  381.5;

// ----------------------------------------------------------
// LDT_START_MOLCH_S1 STARTTASTER AB SIRUPKUECHE
// ----------------------------------------------------------
      SET   ;
      =     DB2981.DBX  441.4;
      =     DB2981.DBX  441.5;

// ----------------------------------------------------------
// LANG_STOER_DOSIERUNG RUECKMELDUNG VON LANG AN TU
// ----------------------------------------------------------
      CLR   ;
//      =     "U098SpID".LANG_STOER_DOSIERUNG.EAl
//      =     "U098SpID".LANG_STOER_DOSIERUNG.Pre

// ----------------------------------------------------------
// LiveBit
// ----------------------------------------------------------
      SET   ;
      =     DB2981.DBX  561.4;
      =     DB2981.DBX  561.5;

NETWORK
TITLE =Messages

      NOP   0;

// ----------------------------------------------------------
// msg001 Message 01
// ----------------------------------------------------------
      SET   ;
      R     DB2987.DBX   80.7;
      =     DB2987.DBX   81.4;

      CLR   ;
      =     DB2987.DBX   82.7;

// ----------------------------------------------------------
// msg002 Message 02
// ----------------------------------------------------------
      SET   ;
      R     DB2987.DBX  140.7;
      =     DB2987.DBX  141.4;

      CLR   ;
      =     DB2987.DBX  142.7;

NETWORK
TITLE =Sequence organisation

      CLR   ;
      =     M    122.2;

// SFM supply ----------------------------------------------------------------

// analog value to SFM Produkttemp. Erhitzer -----------------------
      L     DB2983.DBD  146;
      T     DB1981.DBD 1122; // !!! insert correct SFM !!!

// analog value to SFM Erhitzungsregelung Heisswasser -----------------------
      L     DB2983.DBD  266;
      T     DB1981.DBD 1122; // !!! insert correct SFM !!!

// analog value to SFM Produkttemp. Kühler -----------------------
      L     DB2983.DBD  386;
      T     DB1981.DBD 1122; // !!! insert correct SFM !!!

// analog value to SFM Produkteintrittstemp. -----------------------
      L     DB2983.DBD  506;
      T     DB1981.DBD 1122; // !!! insert correct SFM !!!

// sequencer ----------------------------------------------------------------
      A     DB1983.DBX   43.1;
      S     DB1983.DBX   97.3;

      CALL FC    40 (
           UnitNo                   := #UnitNo);

NETWORK
TITLE =Auto / Manual

      SET   ;
      AN    M    122.2;
      JC    MODE;
      AN    M    120.1;

// assign actuator mode
      AN    M    120.1;
      =     DB2980.DBX  105.4;
      =     DB2980.DBX  185.4;
      =     DB2980.DBX  265.4;
      =     DB2980.DBX  345.4;
      =     DB2980.DBX  425.4;
      =     DB2980.DBX  505.4;
      =     DB2980.DBX  585.4;
      =     DB2980.DBX  665.4;



MODE: SET   ;

NETWORK
TITLE =KZE_RBTR SIGNAL AN SCHMIDT KZE SK
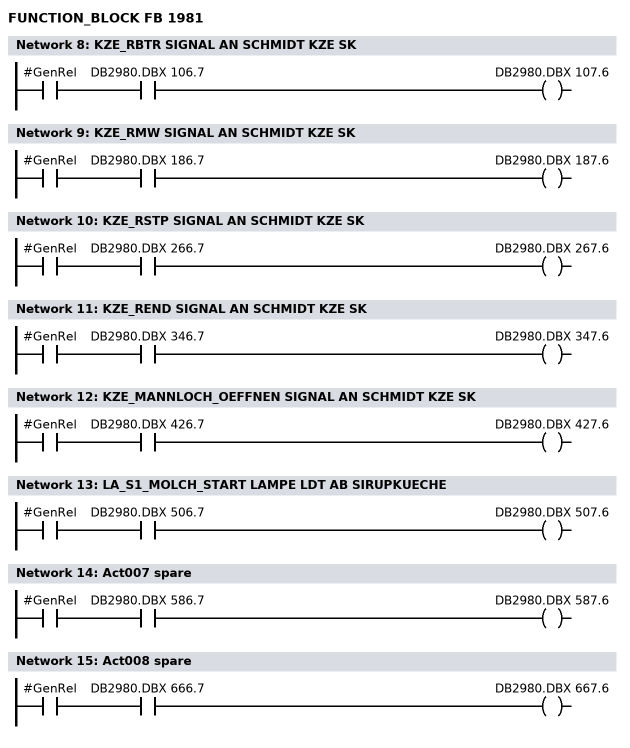

      A     #GenRel;
      A     DB2980.DBX  106.7;
      =     DB2980.DBX  107.6;
NETWORK
TITLE =KZE_RMW SIGNAL AN SCHMIDT KZE SK

      A     #GenRel;
      A     DB2980.DBX  186.7;
      =     DB2980.DBX  187.6;
NETWORK
TITLE =KZE_RSTP SIGNAL AN SCHMIDT KZE SK

      A     #GenRel;
      A     DB2980.DBX  266.7;
      =     DB2980.DBX  267.6;
NETWORK
TITLE =KZE_REND SIGNAL AN SCHMIDT KZE SK

      A     #GenRel;
      A     DB2980.DBX  346.7;
      =     DB2980.DBX  347.6;
NETWORK
TITLE =KZE_MANNLOCH_OEFFNEN SIGNAL AN SCHMIDT KZE SK

      A     #GenRel;
      A     DB2980.DBX  426.7;
      =     DB2980.DBX  427.6;
NETWORK
TITLE =LA_S1_MOLCH_START LAMPE LDT AB SIRUPKUECHE

      A     #GenRel;
      A     DB2980.DBX  506.7;
      =     DB2980.DBX  507.6;
NETWORK
TITLE =Act007 spare

      A     #GenRel;
      A     DB2980.DBX  586.7;
      =     DB2980.DBX  587.6;
NETWORK
TITLE =Act008 spare

      A     #GenRel;
      A     DB2980.DBX  666.7;
      =     DB2980.DBX  667.6;
END_FUNCTION_BLOCK

FUNCTION_BLOCK FB 1990
TITLE =U099: PLC 3 General
FAMILY : BOTEC_F1
NAME : UniA
VERSION : 2.1


VAR_TEMP
  EStopOK : BOOL ;	//auxiliary flag
  CIP : BOOL ;	//CIP Program Selected
  xTmp : BOOL ;	//Temporary Bool(free for general use)
  UnitNo : INT ;	//unit number
  UnitFB : INT ;	//unit expansion FB number
  rTmp : REAL ;	//Temporary REAL (free for general use)
  iTmp : INT ;	//Temporary INT (free for general use)
  dTmp : DINT ;	//Temporary DINT (free for general use)
END_VAR
BEGIN
NETWORK
TITLE =general

      CLR   ;
      =     #xTmp;
      =     #EStopOK;

      L     DB1990.DBW    0;
      T     #UnitNo;
      L     DB1990.DBW    2;
      T     #UnitFB;

NETWORK
TITLE =analog inputs

      NOP   0;
// LIT_ZST AnI 001 Füllstandsanzeige Zitronensäuretank
      CALL FC    24 (
           UnitNo                   := #UnitNo,
           AnIRec                   := DB2993.LIT_ZST,
           ValPer                   := IW   532);

NETWORK
TITLE =Universal value

      NOP   0;
// unv001 UnV 001 Process Status
      CALL FC    27 (
           UnitNo                   := #UnitNo,
           UnVRec                   := DB2995.unv001,
           ValExt                   := DB2995.DBD  234);

// unv002 UnV 002 Universal Value 02
      CALL FC    27 (
           UnitNo                   := #UnitNo,
           UnVRec                   := DB2995.unv002,
           ValExt                   := DB2995.DBD  362);

NETWORK
TITLE =special inputs

      NOP   0;
// NOT_STOP SpI 001 Not-Stop für alle Programme von extern
      CALL FC    14 (
           UnitNo                   := #UnitNo,
           SpIRec                   := DB2991.NOT_STOP,
           SpIBit                   := I      7.2);

// S5_EP1_HAND_EIN_LAUTO SpI 002 SCHALTER PUMPE E.P1
      CALL FC    14 (
           UnitNo                   := #UnitNo,
           SpIRec                   := DB2991.S5_EP1_HAND_EIN_LAUTO,
           SpIBit                   := I     64.2);

// RM_NI_RU_K1 SpI 003
      CALL FC    14 (
           UnitNo                   := #UnitNo,
           SpIRec                   := DB2991.RM_NI_RU_K1,
           SpIBit                   := I     68.6);

// LP_A9_LA10 SpI 006 Lampentest
      CALL FC    14 (
           UnitNo                   := #UnitNo,
           SpIRec                   := DB2991.LP_A9_LA10,
           SpIBit                   := I    258.7);

// GOA_G1 SpI 007 GOA_G1 Schwenkbogen Befüllblock nach Gully
      CALL FC    14 (
           UnitNo                   := #UnitNo,
           SpIRec                   := DB2991.GOA_G1,
           SpIBit                   := I    312.1);

// U99_SpI008 SpI 008 spare
//      CALL  "SI1"
//       UnitNo:=#UnitNo
//       SpIRec:="U099SpID".U99_SpI008
//       SpIBit:=#xTmp

NETWORK
TITLE =messages

      NOP   0;
// msg001 Msg 001 Message 01
      CALL FC    16 (
           UnitNo                   := #UnitNo,
           MsgRec                   := DB2997.msg001,
           MsgBit                   := DB2997.DBX   82.7);

// msg002 Msg 002 Message 02
      CALL FC    16 (
           UnitNo                   := #UnitNo,
           MsgRec                   := DB2997.msg002,
           MsgBit                   := DB2997.DBX  142.7);

NETWORK
TITLE =unit supply

      UC    FB [#UnitFB];

NETWORK
TITLE =RS_GV1
// Act 001
// Box           : Ventilinsel 4
// Input address : I337.5
// Output address: Q337.5
      CALL FC    70 (
           UnitNo                   := #UnitNo,
           ActRec                   := DB2990.RS_GV1,
           Typ                      := 1,
           FBa                      := #xTmp,
           FBa2                     := I    337.5,
           Out                      := Q    337.5);

NETWORK
TITLE =U99_Act003  Tank Emptying CIP Drain
// Act 003
// Box           :
// Output address: #xtmp
      CALL FC    70 (
           UnitNo                   := #UnitNo,
           ActRec                   := DB2990.U99_Act003,
           Typ                      := 0,
           FBa                      := #xTmp,
           FBa2                     := #xTmp,
           Out                      := #xTmp);

END_FUNCTION_BLOCK

FUNCTION_BLOCK FB 1991
TITLE =U099: PLC 3 General
FAMILY : BOTEC_F1
NAME : UniE
VERSION : 1.2


VAR_TEMP
  CIP : BOOL ;	//CIP active
  UNIM : BOOL ;	//Unit Not In Maintenance
  GenRel : BOOL ;	//general OK (emergency and maintenance OK)
  EStopOK : BOOL ;	//emergency OK
  UnitNo : INT ;	//unit number
  xTmp : BOOL ;	//Temporary Bool
  iTmp : INT ;	//Temporary INT
  rTmp : REAL ;	//Temporary REAL
  dTmp : DINT ;	//Temporary DINT (free for general use)
  RetValInt : INT ;	//return value
END_VAR
BEGIN
NETWORK
TITLE =General

      SET   ;
// Simulation ---------------------------------------------------------------
      A     DB1991.DBX 1357.7;
      CC    FB  1999; // "U099Sim"
      A     DB1991.DBX   17.3;
      =     DB1991.DBX 1357.7; //Help bit for simulation

// get unit number ----------------------------------------------------------
      L     DB1990.DBW    0;
      T     #UnitNo;

// CIP ----------------------------------------------------------------------
      L     DB1991.DBD   54;
      L     0;
      <D    ;
      =     #CIP;

// emergency OK -------------------------------------------------------------
      A     DB1995.DBX   27.0; //Emergency Stop OK
      =     #EStopOK;

// Write Unit in Maintenance ------------------------------------------------

      AN    DB1991.DBX   69.7;
      =     #UNIM;

// emergency and maintenance OK ---------------------------------------------
      A     #EStopOK;
      A     #UNIM;
      =     #GenRel;

// communication ------------------------------------------------------------
      UC    FB  1995; // U099Com

NETWORK
TITLE =Analog Inputs

      NOP   0;

// ----------------------------------------------------------
// LIT_ZST Füllstandsanzeige Zitronensäuretank
// ----------------------------------------------------------
      L     DB1991.DBD 1118; // !!! insert correct SFM !!!
      T     DB2993.DBD  238;

      SET   ;
      =     DB2993.DBX  141.5;

NETWORK
TITLE =Universal Value

      NOP   0;

// ----------------------------------------------------------
// unv001 Process Status
// ----------------------------------------------------------
// process value to UnV
//      L     0.000000e+000
//      T     "U099UnVD".unv001.ValExt

// ----------------------------------------------------------
// unv002 Universal Value 02
// ----------------------------------------------------------
// process value to UnV
//      L     0.000000e+000
//      T     "U099UnVD".unv002.ValExt

NETWORK
TITLE =Special Input

      NOP   0;

// ----------------------------------------------------------
// NOT_STOP Not-Stop für alle Programme von extern
// ----------------------------------------------------------
      SET   ;
      =     DB2991.DBX   81.4;
      =     DB2991.DBX   81.5;

// ----------------------------------------------------------
// S5_EP1_HAND_EIN_LAUTO SCHALTER PUMPE E.P1
// ----------------------------------------------------------
      SET   ;
      =     DB2991.DBX  141.4;
      =     DB2991.DBX  141.5;

// ----------------------------------------------------------
// RM_NI_RU_K1
// ----------------------------------------------------------
      SET   ;
      =     DB2991.DBX  201.4;
      =     DB2991.DBX  201.5;

// ----------------------------------------------------------
// GOA_SKP1 GOA
// ----------------------------------------------------------
      SET   ;
      =     DB2991.DBX  261.4;
      =     DB2991.DBX  261.5;

// ----------------------------------------------------------
// GOA_SRGV GOA Molchw. Gully
// ----------------------------------------------------------
      SET   ;
      =     DB2991.DBX  321.4;
      =     DB2991.DBX  321.5;

// ----------------------------------------------------------
// LP_A9_LA10 Lampentest
// ----------------------------------------------------------
      SET   ;
      =     DB2991.DBX  381.4;
      =     DB2991.DBX  381.5;

// ----------------------------------------------------------
// GOA_G1 GOA_G1 Schwenkbogen Befüllblock nach Gully
// ----------------------------------------------------------
      SET   ;
      =     DB2991.DBX  441.4;
      =     DB2991.DBX  441.5;

// ----------------------------------------------------------
// U99_SpI008 Swingbend Filling tank block to CIP2 return
// ----------------------------------------------------------
      SET   ;
      =     DB2991.DBX  501.4;
      =     DB2991.DBX  501.5;

NETWORK
TITLE =Messages

      NOP   0;

// ----------------------------------------------------------
// msg001 Message 01
// ----------------------------------------------------------
      SET   ;
      R     DB2997.DBX   80.7;
      =     DB2997.DBX   81.4;

      CLR   ;
      =     DB2997.DBX   82.7;

// ----------------------------------------------------------
// msg002 Message 02
// ----------------------------------------------------------
      SET   ;
      R     DB2997.DBX  140.7;
      =     DB2997.DBX  141.4;

      CLR   ;
      =     DB2997.DBX  142.7;

NETWORK
TITLE =Sequence organisation

      CLR   ;
      =     M    122.2;

// SFM supply ----------------------------------------------------------------

// analog value to SFM Füllstandsanzeige Zitronensäuretank -----------------------
      L     DB2993.DBD  146;
      T     DB1991.DBD 1122; // !!! insert correct SFM !!!

// sequencer ----------------------------------------------------------------
      A     DB1993.DBX   43.1;
      S     DB1993.DBX   97.3;

      CALL FC    40 (
           UnitNo                   := #UnitNo);

NETWORK
TITLE =Auto / Manual

      SET   ;
      AN    M    122.2;
      JC    MODE;
      AN    M    120.1;

// assign actuator mode
      AN    M    120.1;
      =     DB2990.DBX  105.4;
      =     DB2990.DBX  185.4;
      =     DB2990.DBX  265.4;



MODE: SET   ;

NETWORK
TITLE =RS_GV1
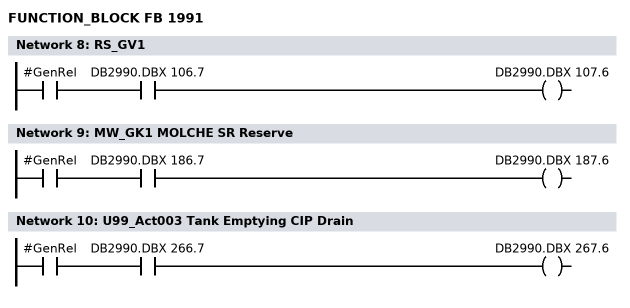

      A     #GenRel;
      A     DB2990.DBX  106.7;
      =     DB2990.DBX  107.6;
NETWORK
TITLE =MW_GK1 MOLCHE SR Reserve

      A     #GenRel;
      A     DB2990.DBX  186.7;
      =     DB2990.DBX  187.6;
NETWORK
TITLE =U99_Act003 Tank Emptying CIP Drain

      A     #GenRel;
      A     DB2990.DBX  266.7;
      =     DB2990.DBX  267.6;
END_FUNCTION_BLOCK

FUNCTION_BLOCK FB 4030
TITLE =U103: Sirup Anlage  3
FAMILY : BOTEC_F1
NAME : U103A
VERSION : 2.1


VAR_TEMP
  EStopOK : BOOL ;	//auxiliary flag
  CIP : BOOL ;	//CIP Program Selected
  xTmp : BOOL ;	//Temporary Bool(free for general use)
  DummyBool : BOOL ;	//Temporary Bool(free for general use)
  UnitNo : INT ;	//unit number
  UnitFB : INT ;	//unit expansion FB number
  rTmp : REAL ;	//Temporary REAL (free for general use)
  iTmp : INT ;	//Temporary INT (free for general use)
  DummyInt : INT ;	//Temporary INT (free for general use)
  dTmp : DINT ;	//Temporary DINT (free for general use)
END_VAR
BEGIN
NETWORK
TITLE =general

      CLR   ;
      =     #xTmp;
      =     #EStopOK;

      L     DB4030.DBW    0;
      T     #UnitNo;
      L     DB4030.DBW    2;
      T     #UnitFB;

NETWORK
TITLE =Universal value

      NOP   0;
// unv001 UnV 001 Process Status
      CALL FC    27 (
           UnitNo                   := #UnitNo,
           UnVRec                   := DB5035.unv001,
           ValExt                   := DB5035.DBD  234);

// unv002 UnV 002 Universal Value 02
      CALL FC    27 (
           UnitNo                   := #UnitNo,
           UnVRec                   := DB5035.unv002,
           ValExt                   := DB5035.DBD  362);

// unv003 UnV 003 Universal Value 03
      CALL FC    27 (
           UnitNo                   := #UnitNo,
           UnVRec                   := DB5035.unv003,
           ValExt                   := DB5035.DBD  490);

// unv004 UnV 004 Universal Value 04
      CALL FC    27 (
           UnitNo                   := #UnitNo,
           UnVRec                   := DB5035.unv004,
           ValExt                   := DB5035.DBD  618);

NETWORK
TITLE =special inputs

      NOP   0;
// GOA_SKEG_31_oben SpI 004 GOA_SKEG_31_oben
      CALL FC    14 (
           UnitNo                   := #UnitNo,
           SpIRec                   := DB5031.GOA_SKEG_31_oben,
           SpIBit                   := I    267.1);

// GOA_SKEG_32_unten SpI 005 GOA_SKEG_32_unten
      CALL FC    14 (
           UnitNo                   := #UnitNo,
           SpIRec                   := DB5031.GOA_SKEG_32_unten,
           SpIBit                   := I    267.2);

// GOA_SKEG_1 SpI 006 GOA_SKEG_1
      CALL FC    14 (
           UnitNo                   := #UnitNo,
           SpIRec                   := DB5031.GOA_SKEG_1,
           SpIBit                   := I    266.7);

// GOA_SKEG_2 SpI 007 GOA_SKEG_2
      CALL FC    14 (
           UnitNo                   := #UnitNo,
           SpIRec                   := DB5031.GOA_SKEG_2,
           SpIBit                   := I    267.0);

// SK_KEG_Molch_Abbruch_DT SpI 008 MOLCH KEG Drucktaste Abbruch Sirupraum
      CALL FC    14 (
           UnitNo                   := #UnitNo,
           SpIRec                   := DB5031.SK_KEG_Molch_Abbruch_DT,
           SpIBit                   := I    264.5);

// SK_KEG_START_Molch_LDT SpI 009 MOLCH KEG L-Drucktaste Start Sirupraum
      CALL FC    14 (
           UnitNo                   := #UnitNo,
           SpIRec                   := DB5031.SK_KEG_START_Molch_LDT,
           SpIBit                   := I    265.0);

// KEG_SK1_Handklappe SpI 010 KEG_SK1_Handklappe
      CALL FC    14 (
           UnitNo                   := #UnitNo,
           SpIRec                   := DB5031.KEG_SK1_Handklappe,
           SpIBit                   := I    266.6);

// GOA_EKEG_31_oben SpI 014 GOA_EKEG_31_oben
      CALL FC    14 (
           UnitNo                   := #UnitNo,
           SpIRec                   := DB5031.GOA_EKEG_31_oben,
           SpIBit                   := I     34.5);

// GOA_EKEG_32_unten SpI 015 GOA_EKEG_32_unten
      CALL FC    14 (
           UnitNo                   := #UnitNo,
           SpIRec                   := DB5031.GOA_EKEG_32_unten,
           SpIBit                   := I     34.6);

// GOA_EKEG_3 SpI 016 GOA_EKEG_3
      CALL FC    14 (
           UnitNo                   := #UnitNo,
           SpIRec                   := DB5031.GOA_EKEG_3,
           SpIBit                   := I     34.3);

// GOA_EKEG_4 SpI 017 GOA_EKEG_4
      CALL FC    14 (
           UnitNo                   := #UnitNo,
           SpIRec                   := DB5031.GOA_EKEG_4,
           SpIBit                   := I     34.4);

// KEG_Freigabe_Molch_SS SpI 018 KEG_Freigabe_Molch_SS
      CALL FC    14 (
           UnitNo                   := #UnitNo,
           SpIRec                   := DB5031.KEG_Freigabe_Molch_SS,
           SpIBit                   := I     35.4);

// KEG_Molch_Start_LDT_I SpI 019 KEG_Molch_Start_LDT
      CALL FC    14 (
           UnitNo                   := #UnitNo,
           SpIRec                   := DB5031.KEG_Molch_Start_LDT_I,
           SpIBit                   := I     34.7);

// KEG_Stop_Molch_DT SpI 020 KEG_Stop_Molch_DT
      CALL FC    14 (
           UnitNo                   := #UnitNo,
           SpIRec                   := DB5031.KEG_Stop_Molch_DT,
           SpIBit                   := I     35.5);

// GOA_EKEG_5 SpI 021 GOA Handklappe am Paneel KEG Anlage (CO2)
      CALL FC    14 (
           UnitNo                   := #UnitNo,
           SpIRec                   := DB5031.GOA_EKEG_5,
           SpIBit                   := I     35.1);

// GOA_KEG_RR1 SpI 022 KEG RR Sirup Kreis 1 Schwenkbogen
      CALL FC    14 (
           UnitNo                   := #UnitNo,
           SpIRec                   := DB5031.GOA_KEG_RR1,
           SpIBit                   := I     94.4);

// KEG_MIXER_BOGEN_22_24 SpI 023 KEG Mixer/KZE Schwenkbogen
      CALL FC    14 (
           UnitNo                   := #UnitNo,
           SpIRec                   := DB5031.KEG_MIXER_BOGEN_22_24,
           SpIBit                   := I    951.3);

// GOA_KEG_RR3 SpI 025 KEG RR Sirup Kreis 3 Schwenkbogen
      CALL FC    14 (
           UnitNo                   := #UnitNo,
           SpIRec                   := DB5031.GOA_KEG_RR3,
           SpIBit                   := I     94.5);

NETWORK
TITLE =messages

      NOP   0;
// msg001 Msg 001 Message 01
      CALL FC    16 (
           UnitNo                   := #UnitNo,
           MsgRec                   := DB5037.msg001,
           MsgBit                   := DB5037.DBX   82.7);

// msg002 Msg 002 Message 02
      CALL FC    16 (
           UnitNo                   := #UnitNo,
           MsgRec                   := DB5037.msg002,
           MsgBit                   := DB5037.DBX  142.7);

// msg003 Msg 003 Message 03
      CALL FC    16 (
           UnitNo                   := #UnitNo,
           MsgRec                   := DB5037.msg003,
           MsgBit                   := DB5037.DBX  202.7);

NETWORK
TITLE =unit supply

      UC    FB [#UnitFB];

NETWORK
TITLE =KEG_MWV1  Ansteuerung KEG_MWV1
// Act 002
// Box           : VS-SRA
// Output address: Q190.0
      CALL FC    70 (
           UnitNo                   := #UnitNo,
           ActRec                   := DB5030.KEG_MWV1,
           Typ                      := 0,
           FBa                      := #xTmp,
           FBa2                     := #xTmp,
           Out                      := Q    190.0);

NETWORK
TITLE =SKEG_V2  Ansteuerung SKEG_V2
// Act 003
// Box           : VS-SRA
// Output address: Q190.1
      CALL FC    70 (
           UnitNo                   := #UnitNo,
           ActRec                   := DB5030.SKEG_V2,
           Typ                      := 0,
           FBa                      := #xTmp,
           FBa2                     := #xTmp,
           Out                      := Q    190.1);

NETWORK
TITLE =SKEG_V31  Ansteuerung SKEG_V31 (ohne RM)
// Act 004
// Box           : VS-SRA
// Output address: Q189.4
      CALL FC    70 (
           UnitNo                   := #UnitNo,
           ActRec                   := DB5030.SKEG_V31,
           Typ                      := 0,
           FBa                      := #xTmp,
           FBa2                     := #xTmp,
           Out                      := Q    189.4);

NETWORK
TITLE =SKEG_V32  Ansteuerung SKEG_V32 (ohne RM)
// Act 005
// Box           : VS-SRA
// Output address: Q189.5
      CALL FC    70 (
           UnitNo                   := #UnitNo,
           ActRec                   := DB5030.SKEG_V32,
           Typ                      := 0,
           FBa                      := #xTmp,
           FBa2                     := #xTmp,
           Out                      := Q    189.5);

NETWORK
TITLE =SKEG_V41  Ansteuerung SKEG_V41
// Act 006
// Box           : VS-SRA
// Output address: Q189.6
      CALL FC    70 (
           UnitNo                   := #UnitNo,
           ActRec                   := DB5030.SKEG_V41,
           Typ                      := 0,
           FBa                      := #xTmp,
           FBa2                     := #xTmp,
           Out                      := Q    189.6);

NETWORK
TITLE =SKEG_V42  Ansteuerung SKEG_V42
// Act 007
// Box           : VS-SRA
// Output address: Q189.7
      CALL FC    70 (
           UnitNo                   := #UnitNo,
           ActRec                   := DB5030.SKEG_V42,
           Typ                      := 0,
           FBa                      := #xTmp,
           FBa2                     := #xTmp,
           Out                      := Q    189.7);

NETWORK
TITLE =SK_KEG_Abbruch_Stoerung  Lampe Abbruch IM SIRUPRAUM
// Act 008
// Box           : AB1SK
// Output address: Q264.7
      CALL FC    70 (
           UnitNo                   := #UnitNo,
           ActRec                   := DB5030.SK_KEG_Abbruch_Stoerung,
           Typ                      := 0,
           FBa                      := #xTmp,
           FBa2                     := #xTmp,
           Out                      := Q    264.7);

NETWORK
TITLE =SK_KEG_Molch_Start_LDT  Lampe Start Molch IM SIRUPRAUM
// Act 009
// Box           : AB1SK
// Output address: Q265.0
      CALL FC    70 (
           UnitNo                   := #UnitNo,
           ActRec                   := DB5030.SK_KEG_Molch_Start_LDT,
           Typ                      := 0,
           FBa                      := #xTmp,
           FBa2                     := #xTmp,
           Out                      := Q    265.0);

NETWORK
TITLE =SK_KEG_Molch_bei_KEG  Lampe Molch an A11 IM SIRUPRAUM
// Act 010
// Box           : AB1SK
// Output address: Q264.5
      CALL FC    70 (
           UnitNo                   := #UnitNo,
           ActRec                   := DB5030.SK_KEG_Molch_bei_KEG,
           Typ                      := 0,
           FBa                      := #xTmp,
           FBa2                     := #xTmp,
           Out                      := Q    264.5);

NETWORK
TITLE =SK_KEG_Molch_in_SK  Lampe Molch im SK IM SIRUPRAUM
// Act 011
// Box           : AB1SK
// Output address: Q264.6
      CALL FC    70 (
           UnitNo                   := #UnitNo,
           ActRec                   := DB5030.SK_KEG_Molch_in_SK,
           Typ                      := 0,
           FBa                      := #xTmp,
           FBa2                     := #xTmp,
           Out                      := Q    264.6);

NETWORK
TITLE =EKEG_V1  EKEG_V1
// Act 012
// Box           : VS-KEG
// Input address : I32.4
// Output address: Q32.4
      CALL FC    70 (
           UnitNo                   := #UnitNo,
           ActRec                   := DB5030.EKEG_V1,
           Typ                      := 1,
           FBa                      := #xTmp,
           FBa2                     := I     32.4,
           Out                      := Q     32.4);

NETWORK
TITLE =EKEG_V2  EKEG_V2
// Act 013
// Box           : VS-KEG
// Input address : I32.5
// Output address: Q32.5
      CALL FC    70 (
           UnitNo                   := #UnitNo,
           ActRec                   := DB5030.EKEG_V2,
           Typ                      := 1,
           FBa                      := #xTmp,
           FBa2                     := I     32.5,
           Out                      := Q     32.5);

NETWORK
TITLE =EKEG_V31_o_RM  EKEG_V31_o_RM
// Act 014
// Box           : VS-KEG
// Output address: Q32.0
      CALL FC    70 (
           UnitNo                   := #UnitNo,
           ActRec                   := DB5030.EKEG_V31_o_RM,
           Typ                      := 0,
           FBa                      := #xTmp,
           FBa2                     := #xTmp,
           Out                      := Q     32.0);

NETWORK
TITLE =EKEG_V32_o_RM  EKEG_V32_o_RM
// Act 015
// Box           : VS-KEG
// Output address: Q32.1
      CALL FC    70 (
           UnitNo                   := #UnitNo,
           ActRec                   := DB5030.EKEG_V32_o_RM,
           Typ                      := 0,
           FBa                      := #xTmp,
           FBa2                     := #xTmp,
           Out                      := Q     32.1);

NETWORK
TITLE =EKEG_V41  EKEG_V41
// Act 016
// Box           : VS-KEG
// Input address : I32.2
// Output address: Q32.2
      CALL FC    70 (
           UnitNo                   := #UnitNo,
           ActRec                   := DB5030.EKEG_V41,
           Typ                      := 1,
           FBa                      := #xTmp,
           FBa2                     := I     32.2,
           Out                      := Q     32.2);

NETWORK
TITLE =EKEG_V42  EKEG_V42
// Act 017
// Box           : VS-KEG
// Input address : I32.3
// Output address: Q32.3
      CALL FC    70 (
           UnitNo                   := #UnitNo,
           ActRec                   := DB5030.EKEG_V42,
           Typ                      := 1,
           FBa                      := #xTmp,
           FBa2                     := I     32.3,
           Out                      := Q     32.3);

NETWORK
TITLE =KEG_Molch_Start_LDT  KEG_Molch_Start_LDT
// Act 019
// Box           : VS-KEG
// Output address: Q34.7
      CALL FC    70 (
           UnitNo                   := #UnitNo,
           ActRec                   := DB5030.KEG_Molch_Start_LDT,
           Typ                      := 0,
           FBa                      := #xTmp,
           FBa2                     := #xTmp,
           Out                      := Q     34.7);

NETWORK
TITLE =Molch ist unterwegs (Mixer)


      CALL FC    70 (
           UnitNo                   := #UnitNo,
           ActRec                   := DB5030.Act20,
           Typ                      := 0,
           FBa                      := #xTmp,
           FBa2                     := #xTmp,
           Out                      := Q    947.6);

NETWORK
TITLE =Molch in Endposition (Mixer)


      CALL FC    70 (
           UnitNo                   := #UnitNo,
           ActRec                   := DB5030.Act21,
           Typ                      := 0,
           FBa                      := #xTmp,
           FBa2                     := #xTmp,
           Out                      := Q    946.5);

NETWORK
TITLE =A3_Schwenkbogen  "1"=CIP  "0"=Produktion
// Act 028
// Box           : Sirup
// Output address: DB_SEND_DOEHLER.Anlage3.Schwenkbogen
      CALL FC    70 (
           UnitNo                   := #UnitNo,
           ActRec                   := DB5030.A3_Schwenkbogen,
           Typ                      := 0,
           FBa                      := #xTmp,
           FBa2                     := #xTmp,
           Out                      := DB404.DBX   45.0);

NETWORK
TITLE =KEG_Pos_Molch  KEG_Pos_Molch
// Act 030
// Box           : VS-KEG
// Output address: Q34.4
      CALL FC    70 (
           UnitNo                   := #UnitNo,
           ActRec                   := DB5030.KEG_Pos_Molch,
           Typ                      := 0,
           FBa                      := #xTmp,
           FBa2                     := #xTmp,
           Out                      := Q     34.4);

NETWORK
TITLE =KEG_Laufzeit_Molch  KEG_Laufzeit_Molch
// Act 031
// Box           : VS-KEG
// Output address: Q34.5
      CALL FC    70 (
           UnitNo                   := #UnitNo,
           ActRec                   := DB5030.KEG_Laufzeit_Molch,
           Typ                      := 0,
           FBa                      := #xTmp,
           FBa2                     := #xTmp,
           Out                      := Q     34.5);

NETWORK
TITLE =KEG_Temperatur_erreicht  KEG_Temperatur_erreicht
// Act 032
// Box           : VS-KEG
// Output address: Q34.6
      CALL FC    70 (
           UnitNo                   := #UnitNo,
           ActRec                   := DB5030.KEG_Temperatur_erreicht,
           Typ                      := 0,
           FBa                      := #xTmp,
           FBa2                     := #xTmp,
           Out                      := Q     34.6);

NETWORK
TITLE =A3_Molch_Sirup  "1"=Molch ist im Sirupraum
// Act 046
// Box           : Sirup
// Output address: DB_SEND_DOEHLER.Anlage3.Molch_Sirup
      CALL FC    70 (
           UnitNo                   := #UnitNo,
           ActRec                   := DB5030.A3_Molch_Sirup,
           Typ                      := 0,
           FBa                      := #xTmp,
           FBa2                     := #xTmp,
           Out                      := DB404.DBX   44.0);

NETWORK
TITLE =A3_Molch_Anlage  "1"=Molch ist an der Anlage
// Act 047
// Box           : Sirup
// Output address: DB_SEND_DOEHLER.Anlage3.Molch_Anlage
      CALL FC    70 (
           UnitNo                   := #UnitNo,
           ActRec                   := DB5030.A3_Molch_Anlage,
           Typ                      := 0,
           FBa                      := #xTmp,
           FBa2                     := #xTmp,
           Out                      := DB404.DBX   44.1);

NETWORK
TITLE =A3_Molch_PRO  "1"=Molch ist bereit für Produktion
// Act 048
// Box           : Sirup
// Output address: DB_SEND_DOEHLER.Anlage3.Molch_PRO
      CALL FC    70 (
           UnitNo                   := #UnitNo,
           ActRec                   := DB5030.A3_Molch_PRO,
           Typ                      := 0,
           FBa                      := #xTmp,
           FBa2                     := #xTmp,
           Out                      := DB404.DBX   44.2);

NETWORK
TITLE =A3_Molch_CIP  "1"=Molch ist bereit für CIP
// Act 049
// Box           : Sirup
// Output address: DB_SEND_DOEHLER.Anlage3.Molch_CIP
      CALL FC    70 (
           UnitNo                   := #UnitNo,
           ActRec                   := DB5030.A3_Molch_CIP,
           Typ                      := 0,
           FBa                      := #xTmp,
           FBa2                     := #xTmp,
           Out                      := DB404.DBX   44.3);

NETWORK
TITLE =A3_Sirupanforderung
// Act 050
// Box           : Sirup
// Output address: DB_SEND_DOEHLER.Anlage3.Sirupanforderung
      CALL FC    70 (
           UnitNo                   := #UnitNo,
           ActRec                   := DB5030.A3_Sirupanforderung,
           Typ                      := 0,
           FBa                      := #xTmp,
           FBa2                     := #xTmp,
           Out                      := DB404.DBX   44.4);

END_FUNCTION_BLOCK

FUNCTION_BLOCK FB 4031
TITLE =U103: Sirup Anlage  3
FAMILY : BOTEC_F1
NAME : U103E
VERSION : 1.2


VAR_TEMP
  CIP : BOOL ;	//CIP active
  UNIM : BOOL ;	//Unit Not In Maintenance
  GenRel : BOOL ;	//general OK (emergency and maintenance OK)
  EStopOK : BOOL ;	//emergency OK
  UnitNo : INT ;	//unit number
  xTmp : BOOL ;	//Temporary Bool
  iTmp : INT ;	//Temporary INT
  rTmp : REAL ;	//Temporary REAL
  dTmp : DINT ;	//Temporary DINT (free for general use)
  RetValInt : INT ;	//return value
END_VAR
BEGIN
NETWORK
TITLE =General

      SET   ;
// Simulation ---------------------------------------------------------------
      A     DB4031.DBX 1357.7;
      CC    FB  4039; // "U103Sim"
      A     DB4031.DBX   17.3;
      =     DB4031.DBX 1357.7; //Help bit for simulation

// get unit number ----------------------------------------------------------
      L     DB4030.DBW    0;
      T     #UnitNo;

// CIP ----------------------------------------------------------------------
      L     DB4031.DBD   54;
      L     0;
      <D    ;
      =     #CIP;

// emergency OK -------------------------------------------------------------
      A     DB4035.DBX   27.0; //Emergency Stop OK
      =     #EStopOK;

// Write Unit in Maintenance ------------------------------------------------

      AN    DB4031.DBX   69.7;
      =     #UNIM;

// emergency and maintenance OK ---------------------------------------------
      A     #EStopOK;
      A     #UNIM;
      =     #GenRel;

// communication ------------------------------------------------------------
      UC    FB  4035; // U103Com

NETWORK
TITLE =Universal Value

      NOP   0;

// ----------------------------------------------------------
// unv001 Process Status
// ----------------------------------------------------------
// process value to UnV
//      L     0.000000e+000
//      T     "U103UnVD".unv001.ValExt

// ----------------------------------------------------------
// unv002 Universal Value 02
// ----------------------------------------------------------
// process value to UnV
//      L     0.000000e+000
//      T     "U103UnVD".unv002.ValExt

// ----------------------------------------------------------
// unv003 Universal Value 03
// ----------------------------------------------------------
// process value to UnV
//      L     0.000000e+000
//      T     "U103UnVD".unv003.ValExt

// ----------------------------------------------------------
// unv004 Universal Value 04
// ----------------------------------------------------------
// process value to UnV
//      L     0.000000e+000
//      T     "U103UnVD".unv004.ValExt

NETWORK
TITLE =Special Input

      NOP   0;

// ----------------------------------------------------------
// GOA_SKEG_31_oben GOA_SKEG_31_oben
// ----------------------------------------------------------
      SET   ;
      =     DB5031.DBX  261.4;
      =     DB5031.DBX  261.5;

// ----------------------------------------------------------
// GOA_SKEG_32_unten GOA_SKEG_32_unten
// ----------------------------------------------------------
      SET   ;
      =     DB5031.DBX  321.4;
      =     DB5031.DBX  321.5;

// ----------------------------------------------------------
// GOA_SKEG_1 GOA_SKEG_1
// ----------------------------------------------------------
      SET   ;
      =     DB5031.DBX  381.4;
      =     DB5031.DBX  381.5;

// ----------------------------------------------------------
// GOA_SKEG_2 GOA_SKEG_2
// ----------------------------------------------------------
      SET   ;
      =     DB5031.DBX  441.4;
      =     DB5031.DBX  441.5;

// ----------------------------------------------------------
// SK_KEG_Molch_Abbruch_DT MOLCH KEG Drucktaste Abbruch Sirupraum
// ----------------------------------------------------------
      SET   ;
      =     DB5031.DBX  501.4;
      =     DB5031.DBX  501.5;

// ----------------------------------------------------------
// SK_KEG_START_Molch_LDT MOLCH KEG L-Drucktaste Start Sirupraum
// ----------------------------------------------------------
      SET   ;
      =     DB5031.DBX  561.4;
      =     DB5031.DBX  561.5;

// ----------------------------------------------------------
// KEG_SK1_Handklappe KEG_SK1_Handklappe
// ----------------------------------------------------------
      SET   ;
      =     DB5031.DBX  621.4;
      =     DB5031.DBX  621.5;

// ----------------------------------------------------------
// GOA_EKEG_31_oben GOA_EKEG_31_oben
// ----------------------------------------------------------
      SET   ;
      =     DB5031.DBX  861.4;
      =     DB5031.DBX  861.5;

// ----------------------------------------------------------
// GOA_EKEG_32_unten GOA_EKEG_32_unten
// ----------------------------------------------------------
      SET   ;
      =     DB5031.DBX  921.4;
      =     DB5031.DBX  921.5;

// ----------------------------------------------------------
// GOA_EKEG_3 GOA_EKEG_3
// ----------------------------------------------------------
      SET   ;
      =     DB5031.DBX  981.4;
      =     DB5031.DBX  981.5;

// ----------------------------------------------------------
// GOA_EKEG_4 GOA_EKEG_4
// ----------------------------------------------------------
      SET   ;
      =     DB5031.DBX 1041.4;
      =     DB5031.DBX 1041.5;

// ----------------------------------------------------------
// KEG_Freigabe_Molch_SS KEG_Freigabe_Molch_SS
// ----------------------------------------------------------
      SET   ;
      =     DB5031.DBX 1101.4;
      =     DB5031.DBX 1101.5;

// ----------------------------------------------------------
// KEG_Molch_Start_LDT_I KEG_Molch_Start_LDT
// ----------------------------------------------------------
      SET   ;
      =     DB5031.DBX 1161.4;
      =     DB5031.DBX 1161.5;

// ----------------------------------------------------------
// KEG_Stop_Molch_DT KEG_Stop_Molch_DT
// ----------------------------------------------------------
      SET   ;
      =     DB5031.DBX 1221.4;
      =     DB5031.DBX 1221.5;

// ----------------------------------------------------------
// GOA_EKEG_5 GOA Handklappe am Paneel KEG Anlage (CO2)
// ----------------------------------------------------------
      SET   ;
      =     DB5031.DBX 1281.4;
      =     DB5031.DBX 1281.5;

// ----------------------------------------------------------
// GOA_KEG_RR1 KEG RR Sirup Kreis 1 Schwenkbogen
// ----------------------------------------------------------
      SET   ;
      =     DB5031.DBX 1341.4;
      =     DB5031.DBX 1341.5;

// ----------------------------------------------------------
// KEG_MIXER_BOGEN_22_24 KEG Mixer/KZE Schwenkbogen
// ----------------------------------------------------------
      SET   ;
      =     DB5031.DBX 1401.4;
      =     DB5031.DBX 1401.5;

// ----------------------------------------------------------
// GOA_KEG_RR3 KEG RR Sirup Kreis 3 Schwenkbogen
// ----------------------------------------------------------
      SET   ;
      =     DB5031.DBX 1521.4;
      =     DB5031.DBX 1521.5;

NETWORK
TITLE =Messages

      NOP   0;

// ----------------------------------------------------------
// msg001 Message 01
// ----------------------------------------------------------
      SET   ;
      R     DB5037.DBX   80.7;
      =     DB5037.DBX   81.4;

      CLR   ;
      =     DB5037.DBX   82.7;

// ----------------------------------------------------------
// msg002 Message 02
// ----------------------------------------------------------
      SET   ;
      R     DB5037.DBX  140.7;
      =     DB5037.DBX  141.4;

      CLR   ;
      =     DB5037.DBX  142.7;

// ----------------------------------------------------------
// msg003 Message 03
// ----------------------------------------------------------
      SET   ;
      R     DB5037.DBX  200.7;
      =     DB5037.DBX  201.4;

      CLR   ;
      =     DB5037.DBX  202.7;

NETWORK
TITLE =Sequence organisation

      CLR   ;
      =     M    122.2;

// SFM supply ----------------------------------------------------------------

// sequencer ----------------------------------------------------------------
      A     DB4033.DBX   43.1;
      S     DB4033.DBX   97.3;

      CALL FC    40 (
           UnitNo                   := #UnitNo);

NETWORK
TITLE =Auto / Manual

      SET   ;
      AN    M    122.2;
      JC    MODE;
      AN    M    120.1;

// assign actuator mode
      AN    M    120.1;
      =     DB5030.DBX  185.4;
      =     DB5030.DBX  265.4;
      =     DB5030.DBX  345.4;
      =     DB5030.DBX  425.4;
      =     DB5030.DBX  505.4;
      =     DB5030.DBX  585.4;
      =     DB5030.DBX  665.4;
      =     DB5030.DBX  745.4;
      =     DB5030.DBX  825.4;
      =     DB5030.DBX  905.4;
      =     DB5030.DBX  985.4;
      =     DB5030.DBX 1065.4;
      =     DB5030.DBX 1145.4;
      =     DB5030.DBX 1225.4;
      =     DB5030.DBX 1305.4;
      =     DB5030.DBX 1385.4;
      =     DB5030.DBX 1545.4;
      =     DB5030.DBX 2265.4;
      =     DB5030.DBX 2425.4;
      =     DB5030.DBX 2505.4;
      =     DB5030.DBX 2585.4;
      =     DB5030.DBX 3705.4;
      =     DB5030.DBX 3785.4;
      =     DB5030.DBX 3865.4;
      =     DB5030.DBX 3945.4;
      =     DB5030.DBX 4025.4;



MODE: SET   ;

NETWORK
TITLE =KEG_MWV1 Ansteuerung KEG_MWV1
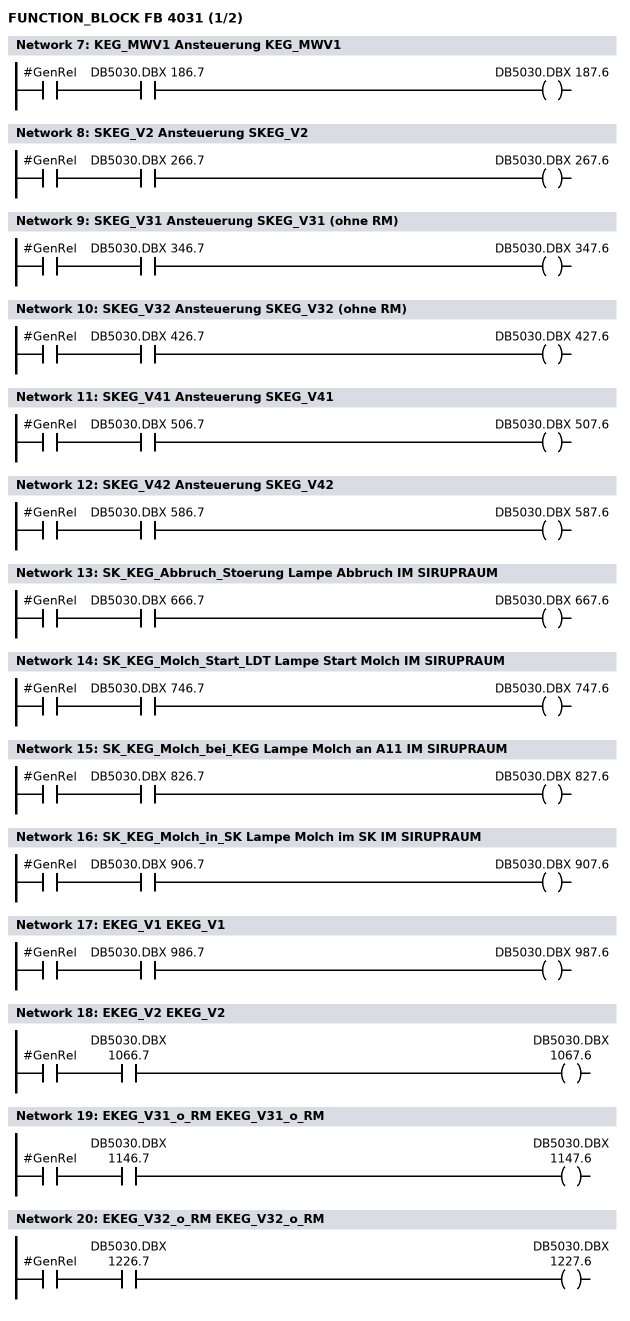

      A     #GenRel;
      A     DB5030.DBX  186.7;
      =     DB5030.DBX  187.6;
NETWORK
TITLE =SKEG_V2 Ansteuerung SKEG_V2

      A     #GenRel;
      A     DB5030.DBX  266.7;
      =     DB5030.DBX  267.6;
NETWORK
TITLE =SKEG_V31 Ansteuerung SKEG_V31 (ohne RM)

      A     #GenRel;
      A     DB5030.DBX  346.7;
      =     DB5030.DBX  347.6;
NETWORK
TITLE =SKEG_V32 Ansteuerung SKEG_V32 (ohne RM)

      A     #GenRel;
      A     DB5030.DBX  426.7;
      =     DB5030.DBX  427.6;
NETWORK
TITLE =SKEG_V41 Ansteuerung SKEG_V41

      A     #GenRel;
      A     DB5030.DBX  506.7;
      =     DB5030.DBX  507.6;
NETWORK
TITLE =SKEG_V42 Ansteuerung SKEG_V42

      A     #GenRel;
      A     DB5030.DBX  586.7;
      =     DB5030.DBX  587.6;
NETWORK
TITLE =SK_KEG_Abbruch_Stoerung Lampe Abbruch IM SIRUPRAUM

      A     #GenRel;
      A     DB5030.DBX  666.7;
      =     DB5030.DBX  667.6;
NETWORK
TITLE =SK_KEG_Molch_Start_LDT Lampe Start Molch IM SIRUPRAUM

      A     #GenRel;
      A     DB5030.DBX  746.7;
      =     DB5030.DBX  747.6;
NETWORK
TITLE =SK_KEG_Molch_bei_KEG Lampe Molch an A11 IM SIRUPRAUM

      A     #GenRel;
      A     DB5030.DBX  826.7;
      =     DB5030.DBX  827.6;
NETWORK
TITLE =SK_KEG_Molch_in_SK Lampe Molch im SK IM SIRUPRAUM

      A     #GenRel;
      A     DB5030.DBX  906.7;
      =     DB5030.DBX  907.6;
NETWORK
TITLE =EKEG_V1 EKEG_V1

      A     #GenRel;
      A     DB5030.DBX  986.7;
      =     DB5030.DBX  987.6;
NETWORK
TITLE =EKEG_V2 EKEG_V2

      A     #GenRel;
      A     DB5030.DBX 1066.7;
      =     DB5030.DBX 1067.6;
NETWORK
TITLE =EKEG_V31_o_RM EKEG_V31_o_RM

      A     #GenRel;
      A     DB5030.DBX 1146.7;
      =     DB5030.DBX 1147.6;
NETWORK
TITLE =EKEG_V32_o_RM EKEG_V32_o_RM

      A     #GenRel;
      A     DB5030.DBX 1226.7;
      =     DB5030.DBX 1227.6;
NETWORK
TITLE =EKEG_V41 EKEG_V41
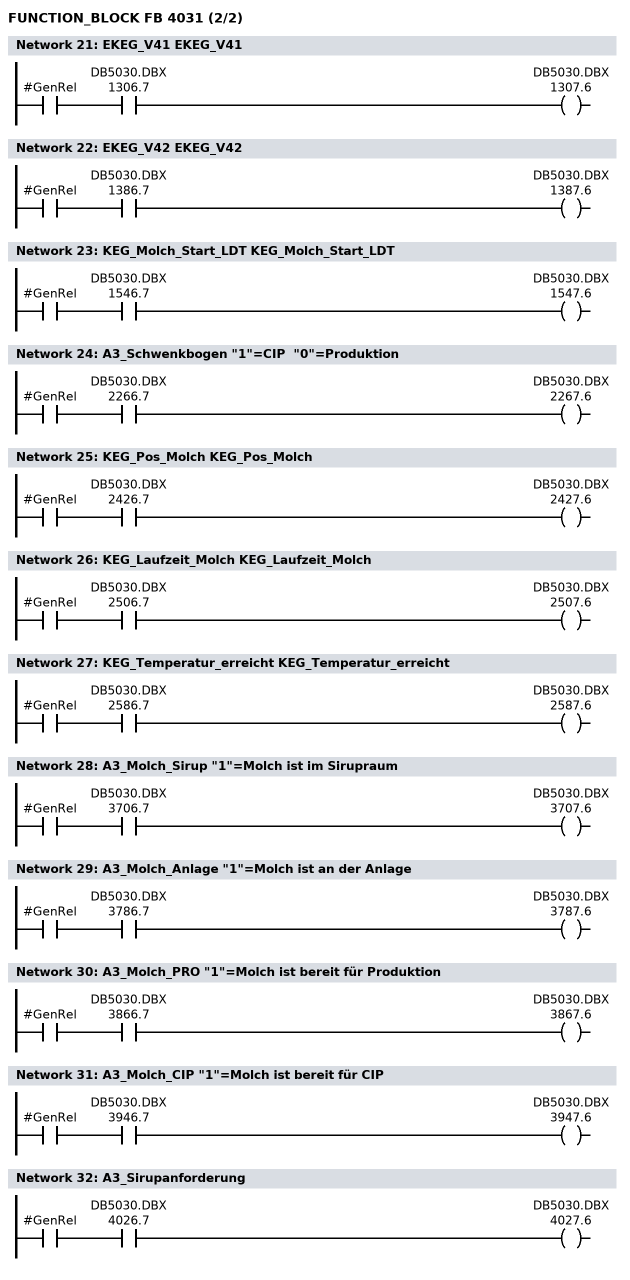

      A     #GenRel;
      A     DB5030.DBX 1306.7;
      =     DB5030.DBX 1307.6;
NETWORK
TITLE =EKEG_V42 EKEG_V42

      A     #GenRel;
      A     DB5030.DBX 1386.7;
      =     DB5030.DBX 1387.6;
NETWORK
TITLE =KEG_Molch_Start_LDT KEG_Molch_Start_LDT

      A     #GenRel;
      A     DB5030.DBX 1546.7;
      =     DB5030.DBX 1547.6;
NETWORK
TITLE =A3_Schwenkbogen "1"=CIP  "0"=Produktion

      A     #GenRel;
      A     DB5030.DBX 2266.7;
      =     DB5030.DBX 2267.6;
NETWORK
TITLE =KEG_Pos_Molch KEG_Pos_Molch

      A     #GenRel;
      A     DB5030.DBX 2426.7;
      =     DB5030.DBX 2427.6;
NETWORK
TITLE =KEG_Laufzeit_Molch KEG_Laufzeit_Molch

      A     #GenRel;
      A     DB5030.DBX 2506.7;
      =     DB5030.DBX 2507.6;
NETWORK
TITLE =KEG_Temperatur_erreicht KEG_Temperatur_erreicht

      A     #GenRel;
      A     DB5030.DBX 2586.7;
      =     DB5030.DBX 2587.6;
NETWORK
TITLE =A3_Molch_Sirup "1"=Molch ist im Sirupraum

      A     #GenRel;
      A     DB5030.DBX 3706.7;
      =     DB5030.DBX 3707.6;
NETWORK
TITLE =A3_Molch_Anlage "1"=Molch ist an der Anlage

      A     #GenRel;
      A     DB5030.DBX 3786.7;
      =     DB5030.DBX 3787.6;
NETWORK
TITLE =A3_Molch_PRO "1"=Molch ist bereit für Produktion

      A     #GenRel;
      A     DB5030.DBX 3866.7;
      =     DB5030.DBX 3867.6;
NETWORK
TITLE =A3_Molch_CIP "1"=Molch ist bereit für CIP

      A     #GenRel;
      A     DB5030.DBX 3946.7;
      =     DB5030.DBX 3947.6;
NETWORK
TITLE =A3_Sirupanforderung

      A     #GenRel;
      A     DB5030.DBX 4026.7;
      =     DB5030.DBX 4027.6;
END_FUNCTION_BLOCK

FUNCTION_BLOCK FB 4050
TITLE =U105: Sirup Anlage  5
FAMILY : BOTEC_F1
NAME : U105A
VERSION : 2.1


VAR_TEMP
  EStopOK : BOOL ;	//auxiliary flag
  CIP : BOOL ;	//CIP Program Selected
  xTmp : BOOL ;	//Temporary Bool(free for general use)
  DummyBool : BOOL ;	//Temporary Bool(free for general use)
  UnitNo : INT ;	//unit number
  UnitFB : INT ;	//unit expansion FB number
  rTmp : REAL ;	//Temporary REAL (free for general use)
  iTmp : INT ;	//Temporary INT (free for general use)
  DummyInt : INT ;	//Temporary INT (free for general use)
  dTmp : DINT ;	//Temporary DINT (free for general use)
END_VAR
BEGIN
NETWORK
TITLE =general

      CLR   ;
      =     #xTmp;
      =     #EStopOK;

      L     DB4050.DBW    0;
      T     #UnitNo;
      L     DB4050.DBW    2;
      T     #UnitFB;

NETWORK
TITLE =Universal value

      NOP   0;
// unv001 UnV 001 Process Status
      CALL FC    27 (
           UnitNo                   := #UnitNo,
           UnVRec                   := DB5055.unv001,
           ValExt                   := DB5055.DBD  234);

// unv002 UnV 002 Universal Value 02
      CALL FC    27 (
           UnitNo                   := #UnitNo,
           UnVRec                   := DB5055.unv002,
           ValExt                   := DB5055.DBD  362);

// unv003 UnV 003 Universal Value 03
      CALL FC    27 (
           UnitNo                   := #UnitNo,
           UnVRec                   := DB5055.unv003,
           ValExt                   := DB5055.DBD  490);

// unv004 UnV 004 Universal Value 04
      CALL FC    27 (
           UnitNo                   := #UnitNo,
           UnVRec                   := DB5055.unv004,
           ValExt                   := DB5055.DBD  618);

NETWORK
TITLE =special inputs

      NOP   0;
// GOA_SA5_31_oben SpI 004 GOA SA5.31 oben Sirupraum
      CALL FC    14 (
           UnitNo                   := #UnitNo,
           SpIRec                   := DB5051.GOA_SA5_31_oben,
           SpIBit                   := I     75.6);

// GOA_SA5_32_unten SpI 005 GOA SA5.32 unten Sirupraum
      CALL FC    14 (
           UnitNo                   := #UnitNo,
           SpIRec                   := DB5051.GOA_SA5_32_unten,
           SpIBit                   := I     75.7);

// GOA_SA5_1 SpI 006 GOA SA5.1 Sirupraum
      CALL FC    14 (
           UnitNo                   := #UnitNo,
           SpIRec                   := DB5051.GOA_SA5_1,
           SpIBit                   := I     75.5);//"GOA_SA5_1"

// GOA_SA5_2 SpI 007 GOA SA5.2 Sirupraum
      CALL FC    14 (
           UnitNo                   := #UnitNo,
           SpIRec                   := DB5051.GOA_SA5_2,
           SpIBit                   := I     75.4);//"GOA_SA5_2"

// SK_A5_Molch_Abbruch_DT SpI 008 MOLCH A5 Drucktaste Abbruch Sirupraum
      CALL FC    14 (
           UnitNo                   := #UnitNo,
           SpIRec                   := DB5051.SK_A5_Molch_Abbruch_DT,
           SpIBit                   := I    181.2);

// SK_A5_START_Molch_LDT SpI 009 MOLCH A5 L-Drucktaste Start Sirupraum
      CALL FC    14 (
           UnitNo                   := #UnitNo,
           SpIRec                   := DB5051.SK_A5_START_Molch_LDT,
           SpIBit                   := I    181.5);

// A5_Sk1_Handklappe SpI 010 GOA Handlappe Anlage 5 SK1 Sirupraum
      CALL FC    14 (
           UnitNo                   := #UnitNo,
           SpIRec                   := DB5051.A5_Sk1_Handklappe,
           SpIBit                   := I     75.3);

// GOA_EA5_31_oben SpI 014 MOLCH A5 GOA EA5.31 oben
      CALL FC    14 (
           UnitNo                   := #UnitNo,
           SpIRec                   := DB5051.GOA_EA5_31_oben,
           SpIBit                   := I    194.5);

// GOA_EA5_32_unten SpI 015 MOLCH A5 GOA EA5.32 unten
      CALL FC    14 (
           UnitNo                   := #UnitNo,
           SpIRec                   := DB5051.GOA_EA5_32_unten,
           SpIBit                   := I    194.6);

// GOA_EA5_3 SpI 016 MOLCH A5 GOA EA5.3
      CALL FC    14 (
           UnitNo                   := #UnitNo,
           SpIRec                   := DB5051.GOA_EA5_3,
           SpIBit                   := I    194.3);

// GOA_EA5_4 SpI 017 MOLCH A5 GOA EA5.4
      CALL FC    14 (
           UnitNo                   := #UnitNo,
           SpIRec                   := DB5051.GOA_EA5_4,
           SpIBit                   := I    194.4);

// A5_SS_FRG_MOLCH SpI 018 Anlage 5 Schlüsselschalter Freigabe Molch
      CALL FC    14 (
           UnitNo                   := #UnitNo,
           SpIRec                   := DB5051.A5_SS_FRG_MOLCH,
           SpIBit                   := I    195.4);

// LDT_Start_A5_MOLCH SpI 019 MOLCH A5 Leuchtdrucktaste Start
      CALL FC    14 (
           UnitNo                   := #UnitNo,
           SpIRec                   := DB5051.LDT_Start_A5_MOLCH,
           SpIBit                   := I    194.7);

// LDT_Stop_A5_MOLCH SpI 020 Anlage 5 Reserve 5
      CALL FC    14 (
           UnitNo                   := #UnitNo,
           SpIRec                   := DB5051.LDT_Stop_A5_MOLCH,
           SpIBit                   := I    195.5);

// A5_K2_Handklappe SpI 021 MOLCH A5 Handklappe K2
      CALL FC    14 (
           UnitNo                   := #UnitNo,
           SpIRec                   := DB5051.A5_K2_Handklappe,
           SpIBit                   := I    195.2);

// GOA501 SpI 022 MOLCH A5 GOA501 --> RR1
      CALL FC    14 (
           UnitNo                   := #UnitNo,
           SpIRec                   := DB5051.GOA501,
           SpIBit                   := I    194.0);

// GOA502 SpI 023 MOLCH A5 GOA502 --> Anlage 5
      CALL FC    14 (
           UnitNo                   := #UnitNo,
           SpIRec                   := DB5051.GOA502,
           SpIBit                   := I    194.1);

// GOA504 SpI 025 Molch A5 GOA504 --> RR3
      CALL FC    14 (
           UnitNo                   := #UnitNo,
           SpIRec                   := DB5051.GOA504,
           SpIBit                   := I    195.3);

NETWORK
TITLE =messages

      NOP   0;
// msg001 Msg 001 Message 01
      CALL FC    16 (
           UnitNo                   := #UnitNo,
           MsgRec                   := DB5057.msg001,
           MsgBit                   := DB5057.DBX   82.7);

// msg002 Msg 002 Message 02
      CALL FC    16 (
           UnitNo                   := #UnitNo,
           MsgRec                   := DB5057.msg002,
           MsgBit                   := DB5057.DBX  142.7);

// msg003 Msg 003 Message 03
      CALL FC    16 (
           UnitNo                   := #UnitNo,
           MsgRec                   := DB5057.msg003,
           MsgBit                   := DB5057.DBX  202.7);

NETWORK
TITLE =unit supply

      UC    FB [#UnitFB];

NETWORK
TITLE =A5_MWV1  MOLCH A5 Ansteuerung MWV1
// Act 002
// Box           : VS-SRA
// Input address : I188.4
// Output address: Q188.4
      CALL FC    70 (
           UnitNo                   := #UnitNo,
           ActRec                   := DB5050.A5_MWV1,
           Typ                      := 1,
           FBa                      := #xTmp,
           FBa2                     := I    188.4,
           Out                      := Q    188.4);

NETWORK
TITLE =SA5_V2  MOLCH SA5 Ansteuerung V2
// Act 003
// Box           : VS-SRA
// Input address : I188.5
// Output address: Q188.5
      CALL FC    70 (
           UnitNo                   := #UnitNo,
           ActRec                   := DB5050.SA5_V2,
           Typ                      := 1,
           FBa                      := #xTmp,
           FBa2                     := I    188.5,
           Out                      := Q    188.5);

NETWORK
TITLE =SA5_V31  MOLCH SA5 Ansteuerung V31 (ohne RM)
// Act 004
// Box           : VS-SRA
// Output address: Q188.0
      CALL FC    70 (
           UnitNo                   := #UnitNo,
           ActRec                   := DB5050.SA5_V31,
           Typ                      := 0,
           FBa                      := #xTmp,
           FBa2                     := #xTmp,
           Out                      := Q    188.0);

NETWORK
TITLE =SA5_V32  MOLCH SA5 Ansteuerung V32 (ohne RM)
// Act 005
// Box           : VS-SRA
// Output address: Q188.1
      CALL FC    70 (
           UnitNo                   := #UnitNo,
           ActRec                   := DB5050.SA5_V32,
           Typ                      := 0,
           FBa                      := #xTmp,
           FBa2                     := #xTmp,
           Out                      := Q    188.1);

NETWORK
TITLE =SA5_V41  MOLCH SA5 Ansteuerung V41
// Act 006
// Box           : VS-SRA
// Input address : I188.2
// Output address: Q188.2
      CALL FC    70 (
           UnitNo                   := #UnitNo,
           ActRec                   := DB5050.SA5_V41,
           Typ                      := 1,
           FBa                      := #xTmp,
           FBa2                     := I    188.2,
           Out                      := Q    188.2);

NETWORK
TITLE =SA5_V42  MOLCH SA5 Ansteuerung V42
// Act 007
// Box           : VS-SRA
// Input address : I188.3
// Output address: Q188.3
      CALL FC    70 (
           UnitNo                   := #UnitNo,
           ActRec                   := DB5050.SA5_V42,
           Typ                      := 1,
           FBa                      := #xTmp,
           FBa2                     := I    188.3,
           Out                      := Q    188.3);

NETWORK
TITLE =SK_A5_Abbruch_L  Anlage 5 Lampe Abbruch IM SIRUPRAUM
// Act 008
// Box           : AB-SK
// Output address: Q181.4
      CALL FC    70 (
           UnitNo                   := #UnitNo,
           ActRec                   := DB5050.SK_A5_Abbruch_L,
           Typ                      := 0,
           FBa                      := #xTmp,
           FBa2                     := #xTmp,
           Out                      := Q    181.4);

